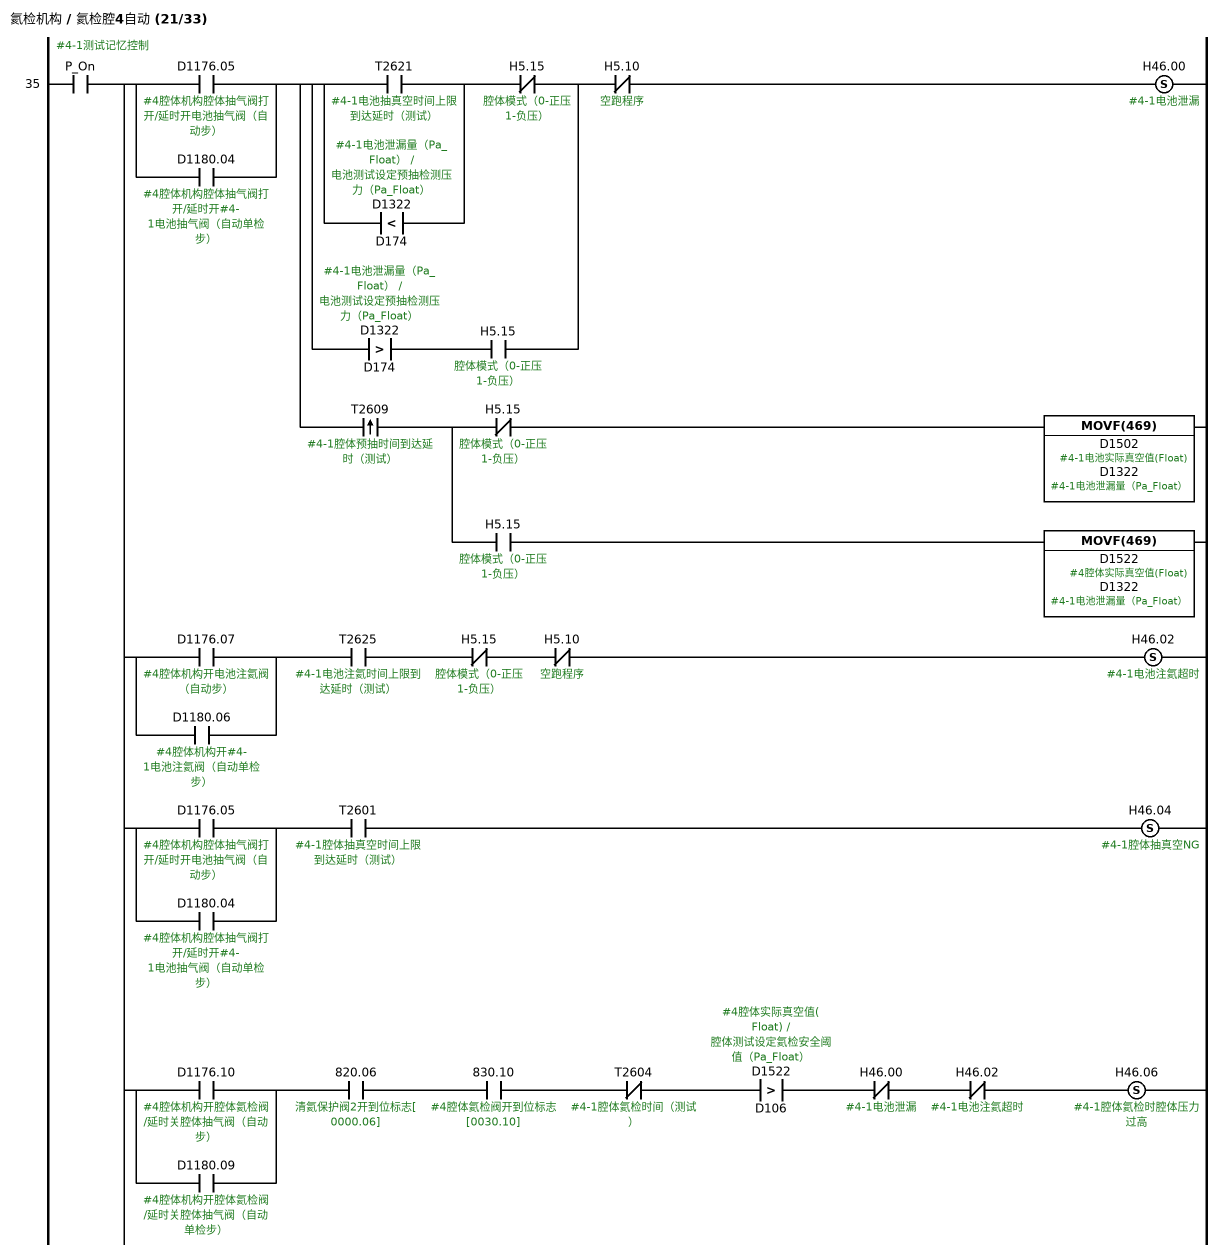
; [picture p360: 氦检机构 / 氦检腔4自动, rungs 35-35]

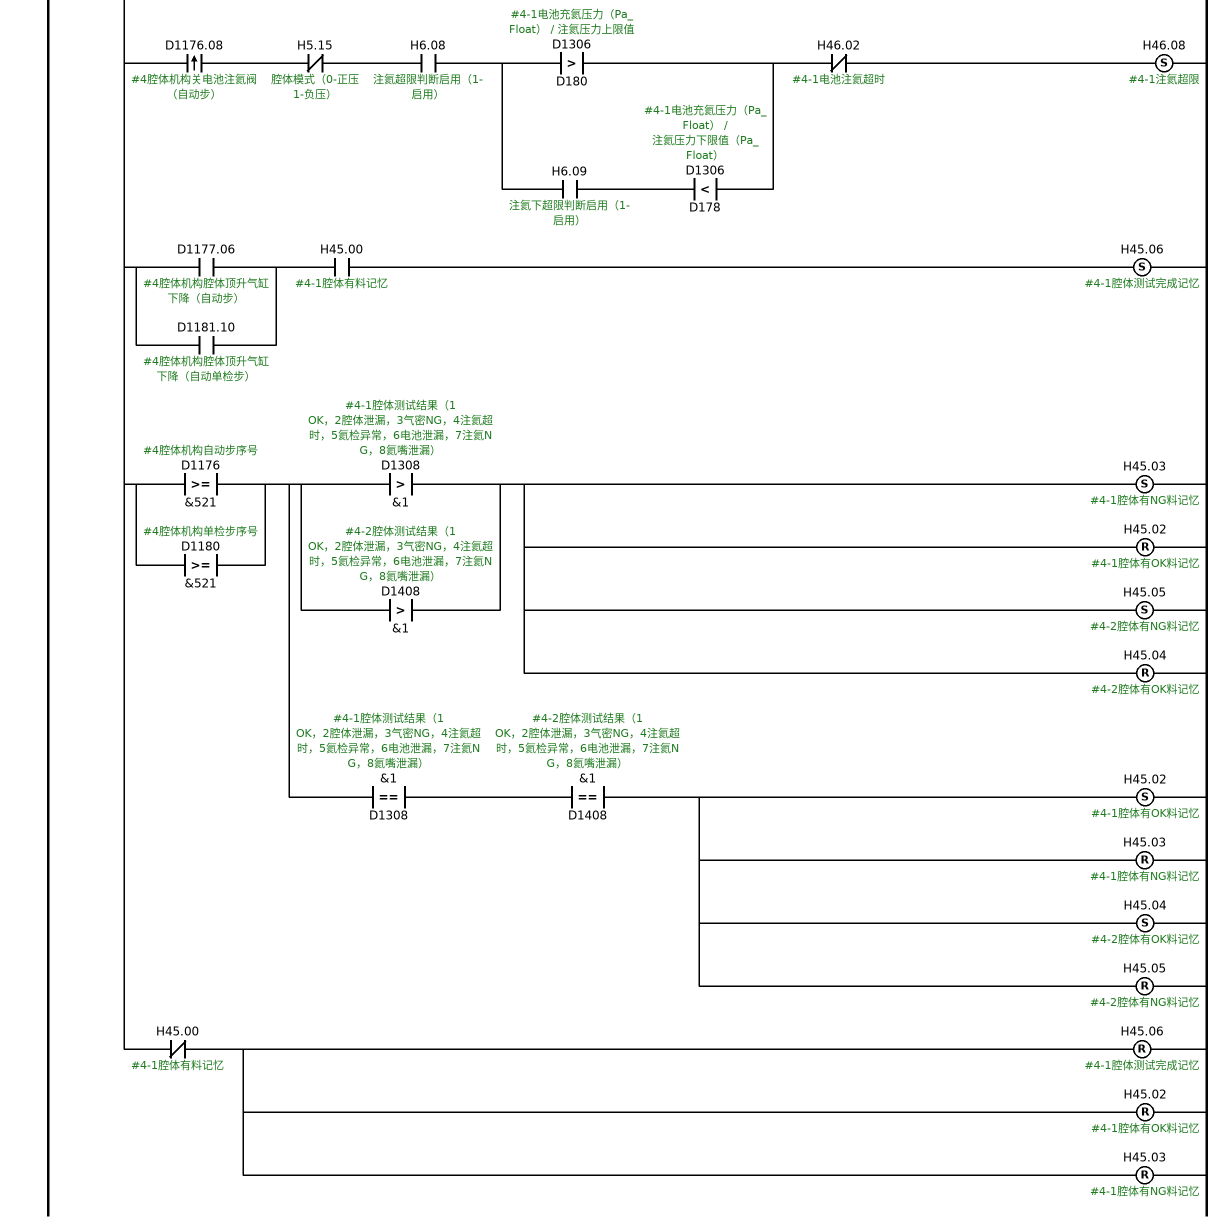
; rung 35: #4-1测试记忆控制
LD P_On
OUT TR0
LD D1176.05  ; #4腔体机构腔体抽气阀打开/延时开电池抽气阀（自动步）
OR D1180.04  ; #4腔体机构腔体抽气阀打开/延时开#4-1电池抽气阀（自动单检步）
ANDLD
OUT TR1
LD T2621  ; #4-1电池抽真空时间上限到达延时（测试）
OR<F(331) D1322 D174  ; #4-1电池泄漏量（Pa_Float）, 电池测试设定预抽检测压力（Pa_Float）
ANDNOT H5.15  ; 腔体模式（0-正压 1-负压）
LD>F(333) D1322 D174  ; #4-1电池泄漏量（Pa_Float）, 电池测试设定预抽检测压力（Pa_Float）
AND H5.15  ; 腔体模式（0-正压 1-负压）
ORLD
ANDLD
ANDNOT H5.10  ; 空跑程序
SET H46.00  ; #4-1电池泄漏
LD TR1
@AND T2609  ; #4-1腔体预抽时间到达延时（测试）
OUT TR1
ANDNOT H5.15  ; 腔体模式（0-正压 1-负压）
MOVF(469) D1502 D1322  ; #4-1电池实际真空值(Float), #4-1电池泄漏量（Pa_Float）
LD TR1
AND H5.15  ; 腔体模式（0-正压 1-负压）
MOVF(469) D1522 D1322  ; #4腔体实际真空值(Float), #4-1电池泄漏量（Pa_Float）
LD TR0
LD D1176.07  ; #4腔体机构开电池注氦阀（自动步）
OR D1180.06  ; #4腔体机构开#4-1电池注氦阀（自动单检步）
ANDLD
AND T2625  ; #4-1电池注氦时间上限到达延时（测试）
ANDNOT H5.15  ; 腔体模式（0-正压 1-负压）
ANDNOT H5.10  ; 空跑程序
SET H46.02  ; #4-1电池注氦超时
LD TR0
LD D1176.05  ; #4腔体机构腔体抽气阀打开/延时开电池抽气阀（自动步）
OR D1180.04  ; #4腔体机构腔体抽气阀打开/延时开#4-1电池抽气阀（自动单检步）
ANDLD
AND T2601  ; #4-1腔体抽真空时间上限到达延时（测试）
SET H46.04  ; #4-1腔体抽真空NG
LD TR0
LD D1176.10  ; #4腔体机构开腔体氦检阀/延时关腔体抽气阀（自动步）
OR D1180.09  ; #4腔体机构开腔体氦检阀/延时关腔体抽气阀（自动单检步）
ANDLD
AND 820.06  ; 清氦保护阀2开到位标志[0000.06]
AND 830.10  ; #4腔体氦检阀开到位标志[0030.10]
ANDNOT T2604  ; #4-1腔体氦检时间（测试）
AND>F(333) D1522 D106  ; #4腔体实际真空值(Float), 腔体测试设定氦检安全阈值（Pa_Float）
ANDNOT H46.00  ; #4-1电池泄漏
ANDNOT H46.02  ; #4-1电池注氦超时
SET H46.06  ; #4-1腔体氦检时腔体压力过高
LD TR0
@AND D1176.08  ; #4腔体机构关电池注氦阀（自动步）
ANDNOT H5.15  ; 腔体模式（0-正压 1-负压）
AND H6.08  ; 注氦超限判断启用（1-启用）
LD>F(333) D1306 D180  ; #4-1电池充氦压力（Pa_Float）, 注氦压力上限值
LD H6.09  ; 注氦下超限判断启用（1-启用）
AND<F(331) D1306 D178  ; #4-1电池充氦压力（Pa_Float）, 注氦压力下限值（Pa_Float）
ORLD
ANDLD
ANDNOT H46.02  ; #4-1电池注氦超时
SET H46.08  ; #4-1注氦超限
LD TR0
LD D1177.06  ; #4腔体机构腔体顶升气缸下降（自动步）
OR D1181.10  ; #4腔体机构腔体顶升气缸下降（自动单检步）
ANDLD
AND H45.00  ; #4-1腔体有料记忆
SET H45.06  ; #4-1腔体测试完成记忆
LD TR0
LD>=L(326) D1176 &521  ; #4腔体机构自动步序号
OR>=L(326) D1180 &521  ; #4腔体机构单检步序号
ANDLD
OUT TR1
LD>(320) D1308 &1  ; #4-1腔体测试结果（1 OK，2腔体泄漏，3气密NG，4注氦超时，5氦检异常，6电池泄漏，7注氦NG，8氦嘴泄漏）
OR>(320) D1408 &1  ; #4-2腔体测试结果（1 OK，2腔体泄漏，3气密NG，4注氦超时，5氦检异常，6电池泄漏，7注氦NG，8氦嘴泄漏）
ANDLD
SET H45.03  ; #4-1腔体有NG料记忆
RSET H45.02  ; #4-1腔体有OK料记忆
SET H45.05  ; #4-2腔体有NG料记忆
RSET H45.04  ; #4-2腔体有OK料记忆
LD TR1
AND=(300) &1 D1308  ; #4-1腔体测试结果（1 OK，2腔体泄漏，3气密NG，4注氦超时，5氦检异常，6电池泄漏，7注氦NG，8氦嘴泄漏）
AND=(300) &1 D1408  ; #4-2腔体测试结果（1 OK，2腔体泄漏，3气密NG，4注氦超时，5氦检异常，6电池泄漏，7注氦NG，8氦嘴泄漏）
SET H45.02  ; #4-1腔体有OK料记忆
RSET H45.03  ; #4-1腔体有NG料记忆
SET H45.04  ; #4-2腔体有OK料记忆
RSET H45.05  ; #4-2腔体有NG料记忆
LD TR0
ANDNOT H45.00  ; #4-1腔体有料记忆
RSET H45.06  ; #4-1腔体测试完成记忆
RSET H45.02  ; #4-1腔体有OK料记忆
RSET H45.03  ; #4-1腔体有NG料记忆

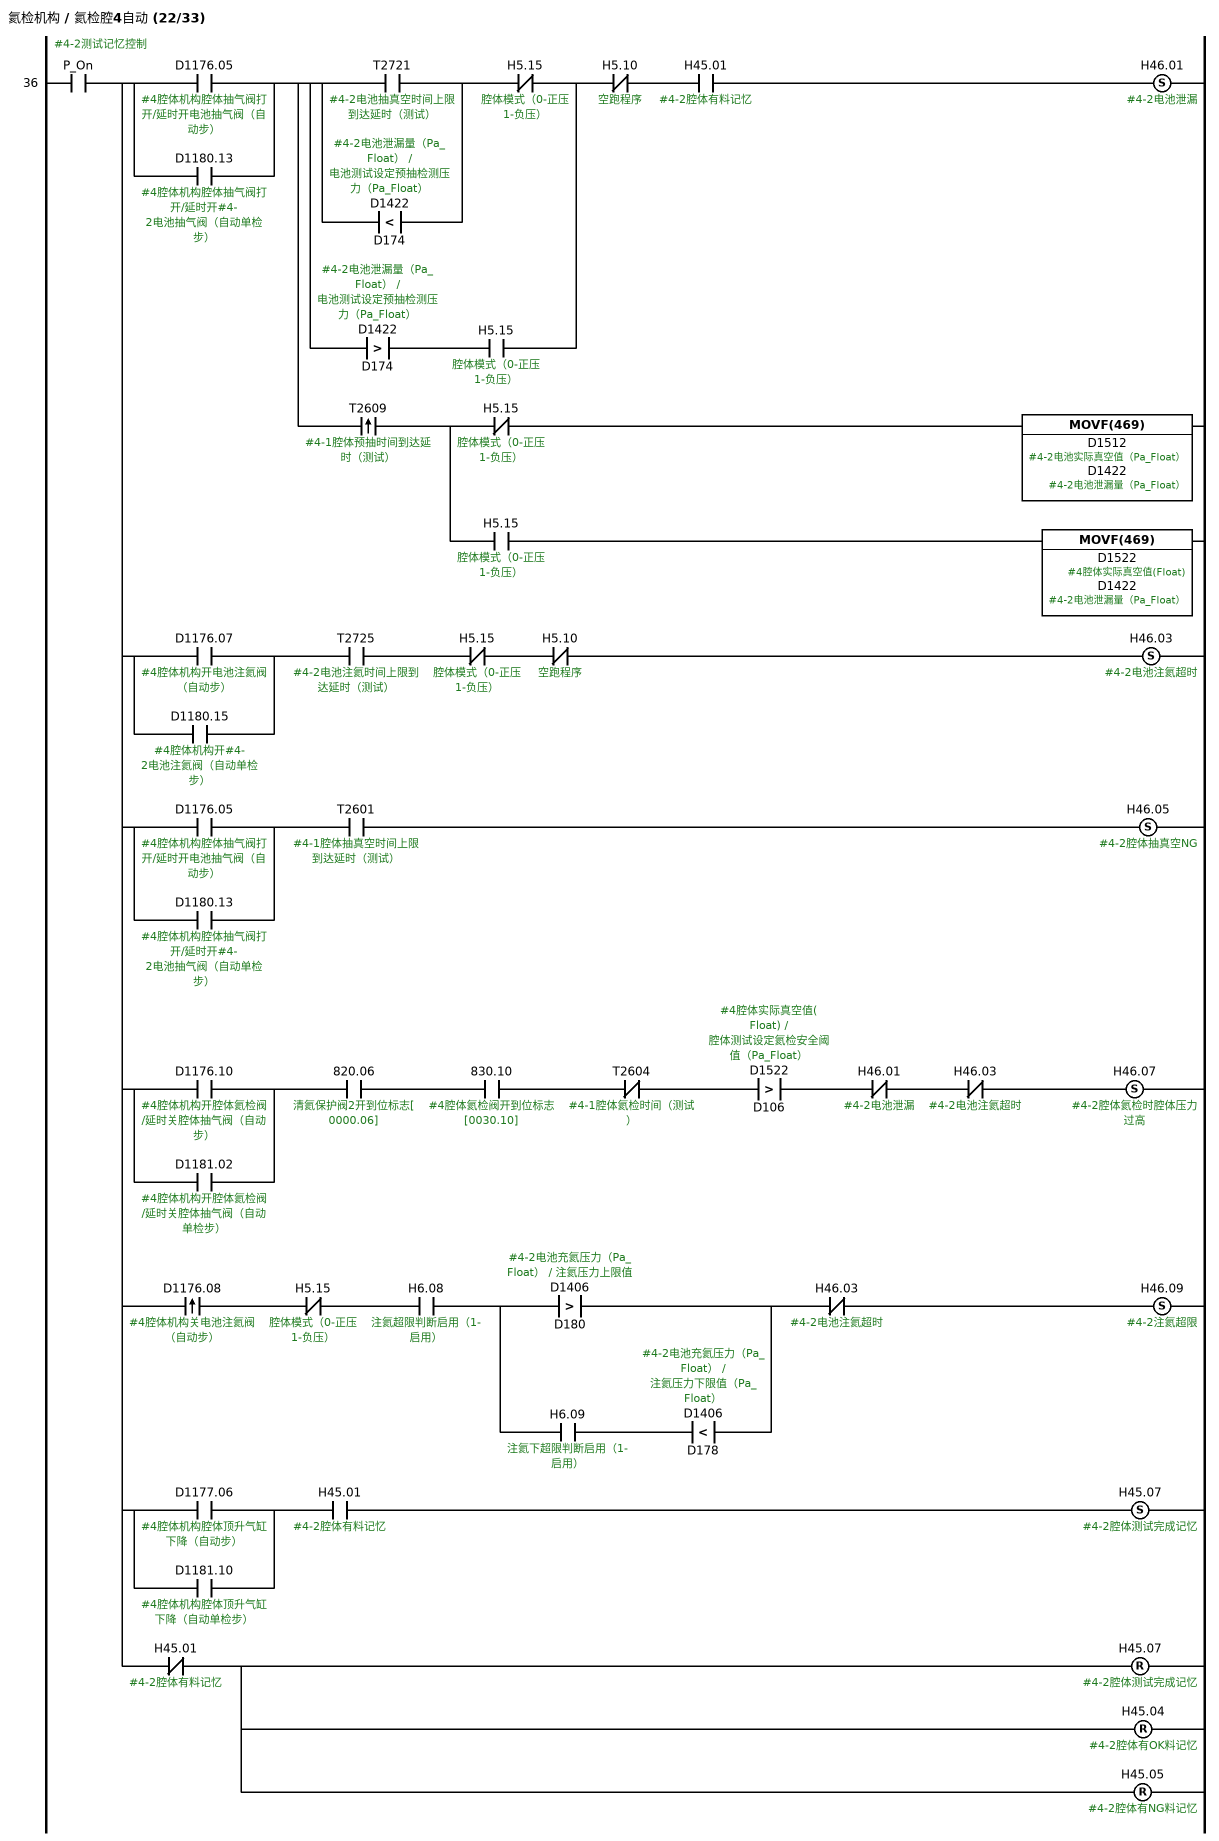
; rung 36: #4-2测试记忆控制
LD P_On
OUT TR0
LD D1176.05  ; #4腔体机构腔体抽气阀打开/延时开电池抽气阀（自动步）
OR D1180.13  ; #4腔体机构腔体抽气阀打开/延时开#4-2电池抽气阀（自动单检步）
ANDLD
OUT TR1
LD T2721  ; #4-2电池抽真空时间上限到达延时（测试）
OR<F(331) D1422 D174  ; #4-2电池泄漏量（Pa_Float）, 电池测试设定预抽检测压力（Pa_Float）
ANDNOT H5.15  ; 腔体模式（0-正压 1-负压）
LD>F(333) D1422 D174  ; #4-2电池泄漏量（Pa_Float）, 电池测试设定预抽检测压力（Pa_Float）
AND H5.15  ; 腔体模式（0-正压 1-负压）
ORLD
ANDLD
ANDNOT H5.10  ; 空跑程序
AND H45.01  ; #4-2腔体有料记忆
SET H46.01  ; #4-2电池泄漏
LD TR1
@AND T2609  ; #4-1腔体预抽时间到达延时（测试）
OUT TR1
ANDNOT H5.15  ; 腔体模式（0-正压 1-负压）
MOVF(469) D1512 D1422  ; #4-2电池实际真空值（Pa_Float）, #4-2电池泄漏量（Pa_Float）
LD TR1
AND H5.15  ; 腔体模式（0-正压 1-负压）
MOVF(469) D1522 D1422  ; #4腔体实际真空值(Float), #4-2电池泄漏量（Pa_Float）
LD TR0
LD D1176.07  ; #4腔体机构开电池注氦阀（自动步）
OR D1180.15  ; #4腔体机构开#4-2电池注氦阀（自动单检步）
ANDLD
AND T2725  ; #4-2电池注氦时间上限到达延时（测试）
ANDNOT H5.15  ; 腔体模式（0-正压 1-负压）
ANDNOT H5.10  ; 空跑程序
SET H46.03  ; #4-2电池注氦超时
LD TR0
LD D1176.05  ; #4腔体机构腔体抽气阀打开/延时开电池抽气阀（自动步）
OR D1180.13  ; #4腔体机构腔体抽气阀打开/延时开#4-2电池抽气阀（自动单检步）
ANDLD
AND T2601  ; #4-1腔体抽真空时间上限到达延时（测试）
SET H46.05  ; #4-2腔体抽真空NG
LD TR0
LD D1176.10  ; #4腔体机构开腔体氦检阀/延时关腔体抽气阀（自动步）
OR D1181.02  ; #4腔体机构开腔体氦检阀/延时关腔体抽气阀（自动单检步）
ANDLD
AND 820.06  ; 清氦保护阀2开到位标志[0000.06]
AND 830.10  ; #4腔体氦检阀开到位标志[0030.10]
ANDNOT T2604  ; #4-1腔体氦检时间（测试）
AND>F(333) D1522 D106  ; #4腔体实际真空值(Float), 腔体测试设定氦检安全阈值（Pa_Float）
ANDNOT H46.01  ; #4-2电池泄漏
ANDNOT H46.03  ; #4-2电池注氦超时
SET H46.07  ; #4-2腔体氦检时腔体压力过高
LD TR0
@AND D1176.08  ; #4腔体机构关电池注氦阀（自动步）
ANDNOT H5.15  ; 腔体模式（0-正压 1-负压）
AND H6.08  ; 注氦超限判断启用（1-启用）
LD>F(333) D1406 D180  ; #4-2电池充氦压力（Pa_Float）, 注氦压力上限值
LD H6.09  ; 注氦下超限判断启用（1-启用）
AND<F(331) D1406 D178  ; #4-2电池充氦压力（Pa_Float）, 注氦压力下限值（Pa_Float）
ORLD
ANDLD
ANDNOT H46.03  ; #4-2电池注氦超时
SET H46.09  ; #4-2注氦超限
LD TR0
LD D1177.06  ; #4腔体机构腔体顶升气缸下降（自动步）
OR D1181.10  ; #4腔体机构腔体顶升气缸下降（自动单检步）
ANDLD
AND H45.01  ; #4-2腔体有料记忆
SET H45.07  ; #4-2腔体测试完成记忆
LD TR0
ANDNOT H45.01  ; #4-2腔体有料记忆
RSET H45.07  ; #4-2腔体测试完成记忆
RSET H45.04  ; #4-2腔体有OK料记忆
RSET H45.05  ; #4-2腔体有NG料记忆

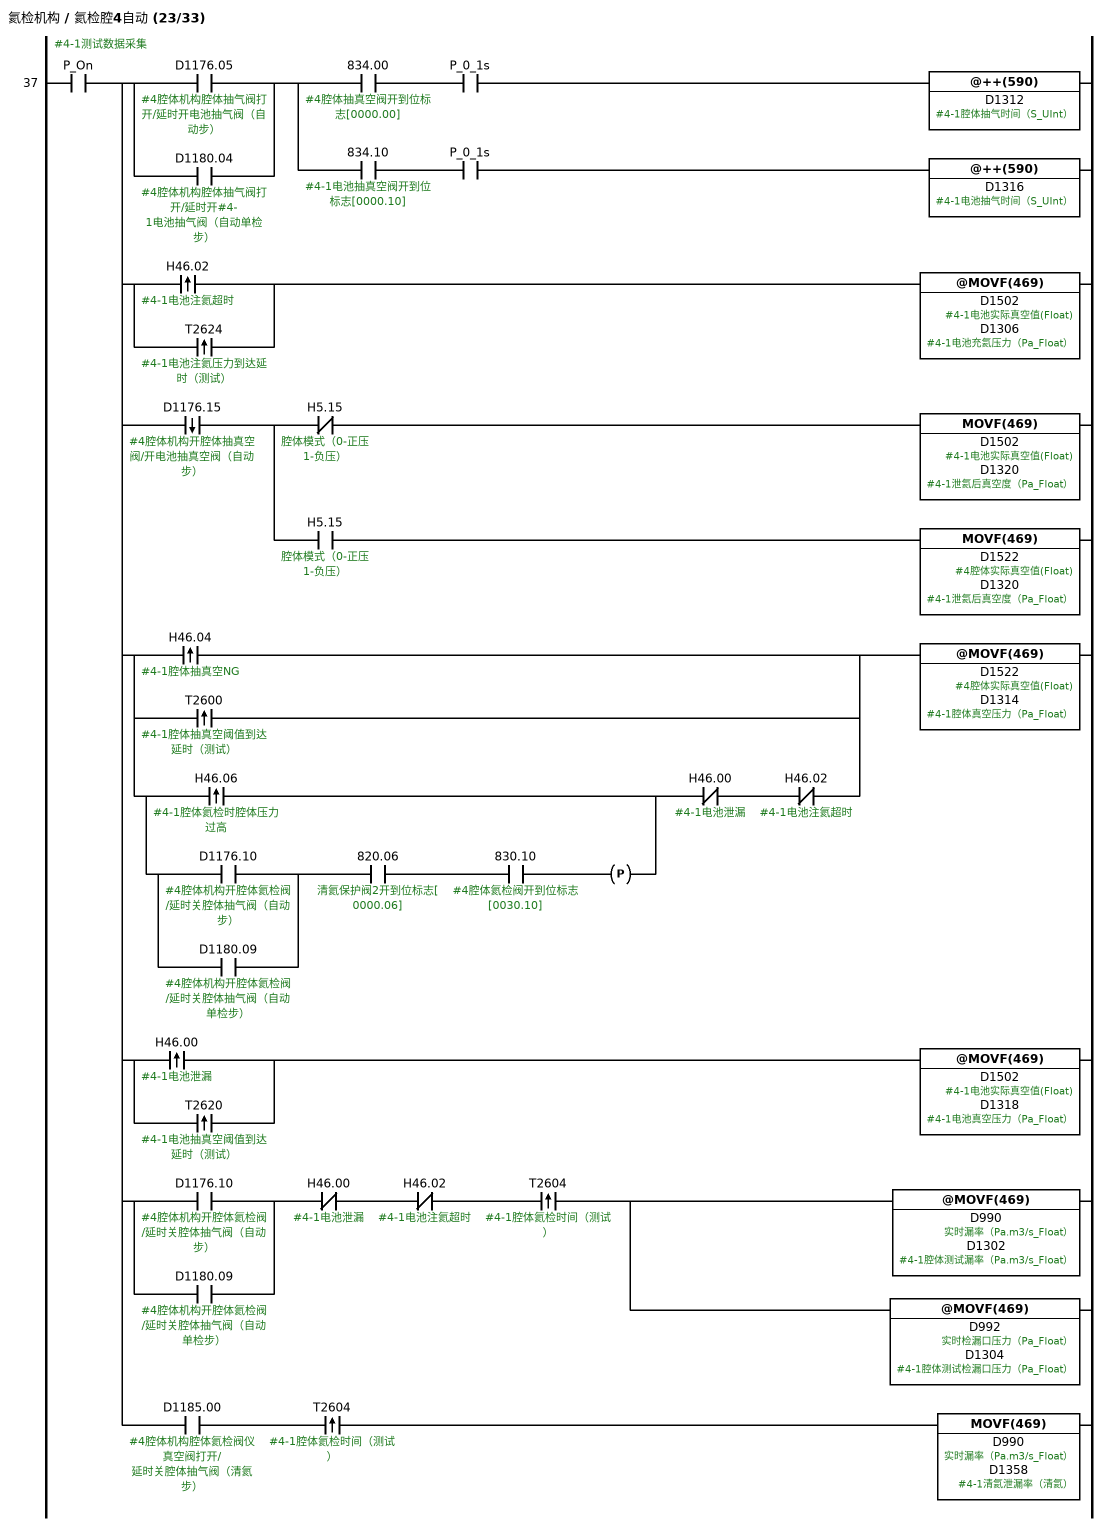
; rung 37: #4-1测试数据采集
LD P_On
OUT TR0
LD D1176.05  ; #4腔体机构腔体抽气阀打开/延时开电池抽气阀（自动步）
OR D1180.04  ; #4腔体机构腔体抽气阀打开/延时开#4-1电池抽气阀（自动单检步）
ANDLD
OUT TR1
AND 834.00  ; #4腔体抽真空阀开到位标志[0000.00]
AND P_0_1s
@++(590) D1312  ; #4-1腔体抽气时间（S_UInt）
LD TR1
AND 834.10  ; #4-1电池抽真空阀开到位标志[0000.10]
AND P_0_1s
@++(590) D1316  ; #4-1电池抽气时间（S_UInt）
LD TR0
@LD H46.02  ; #4-1电池注氦超时
@OR T2624  ; #4-1电池注氦压力到达延时（测试）
ANDLD
@MOVF(469) D1502 D1306  ; #4-1电池实际真空值(Float), #4-1电池充氦压力（Pa_Float）
LD TR0
%AND D1176.15  ; #4腔体机构开腔体抽真空阀/开电池抽真空阀（自动步）
OUT TR1
ANDNOT H5.15  ; 腔体模式（0-正压 1-负压）
MOVF(469) D1502 D1320  ; #4-1电池实际真空值(Float), #4-1泄氦后真空度（Pa_Float）
LD TR1
AND H5.15  ; 腔体模式（0-正压 1-负压）
MOVF(469) D1522 D1320  ; #4腔体实际真空值(Float), #4-1泄氦后真空度（Pa_Float）
LD TR0
@LD H46.04  ; #4-1腔体抽真空NG
@OR T2600  ; #4-1腔体抽真空阈值到达延时（测试）
@LD H46.06  ; #4-1腔体氦检时腔体压力过高
LD D1176.10  ; #4腔体机构开腔体氦检阀/延时关腔体抽气阀（自动步）
OR D1180.09  ; #4腔体机构开腔体氦检阀/延时关腔体抽气阀（自动单检步）
AND 820.06  ; 清氦保护阀2开到位标志[0000.06]
AND 830.10  ; #4腔体氦检阀开到位标志[0030.10]
UP(521)
ORLD
ANDNOT H46.00  ; #4-1电池泄漏
ANDNOT H46.02  ; #4-1电池注氦超时
ORLD
ANDLD
@MOVF(469) D1522 D1314  ; #4腔体实际真空值(Float), #4-1腔体真空压力（Pa_Float）
LD TR0
@LD H46.00  ; #4-1电池泄漏
@OR T2620  ; #4-1电池抽真空阈值到达延时（测试）
ANDLD
@MOVF(469) D1502 D1318  ; #4-1电池实际真空值(Float), #4-1电池真空压力（Pa_Float）
LD TR0
LD D1176.10  ; #4腔体机构开腔体氦检阀/延时关腔体抽气阀（自动步）
OR D1180.09  ; #4腔体机构开腔体氦检阀/延时关腔体抽气阀（自动单检步）
ANDLD
ANDNOT H46.00  ; #4-1电池泄漏
ANDNOT H46.02  ; #4-1电池注氦超时
@AND T2604  ; #4-1腔体氦检时间（测试）
@MOVF(469) D990 D1302  ; 实时漏率（Pa.m3/s_Float）, #4-1腔体测试漏率（Pa.m3/s_Float）
@MOVF(469) D992 D1304  ; 实时检漏口压力（Pa_Float）, #4-1腔体测试检漏口压力（Pa_Float）
LD TR0
AND D1185.00  ; #4腔体机构腔体氦检阀仪真空阀打开/延时关腔体抽气阀（清氦步）
@AND T2604  ; #4-1腔体氦检时间（测试）
MOVF(469) D990 D1358  ; 实时漏率（Pa.m3/s_Float）, #4-1清氦泄漏率（清氦）

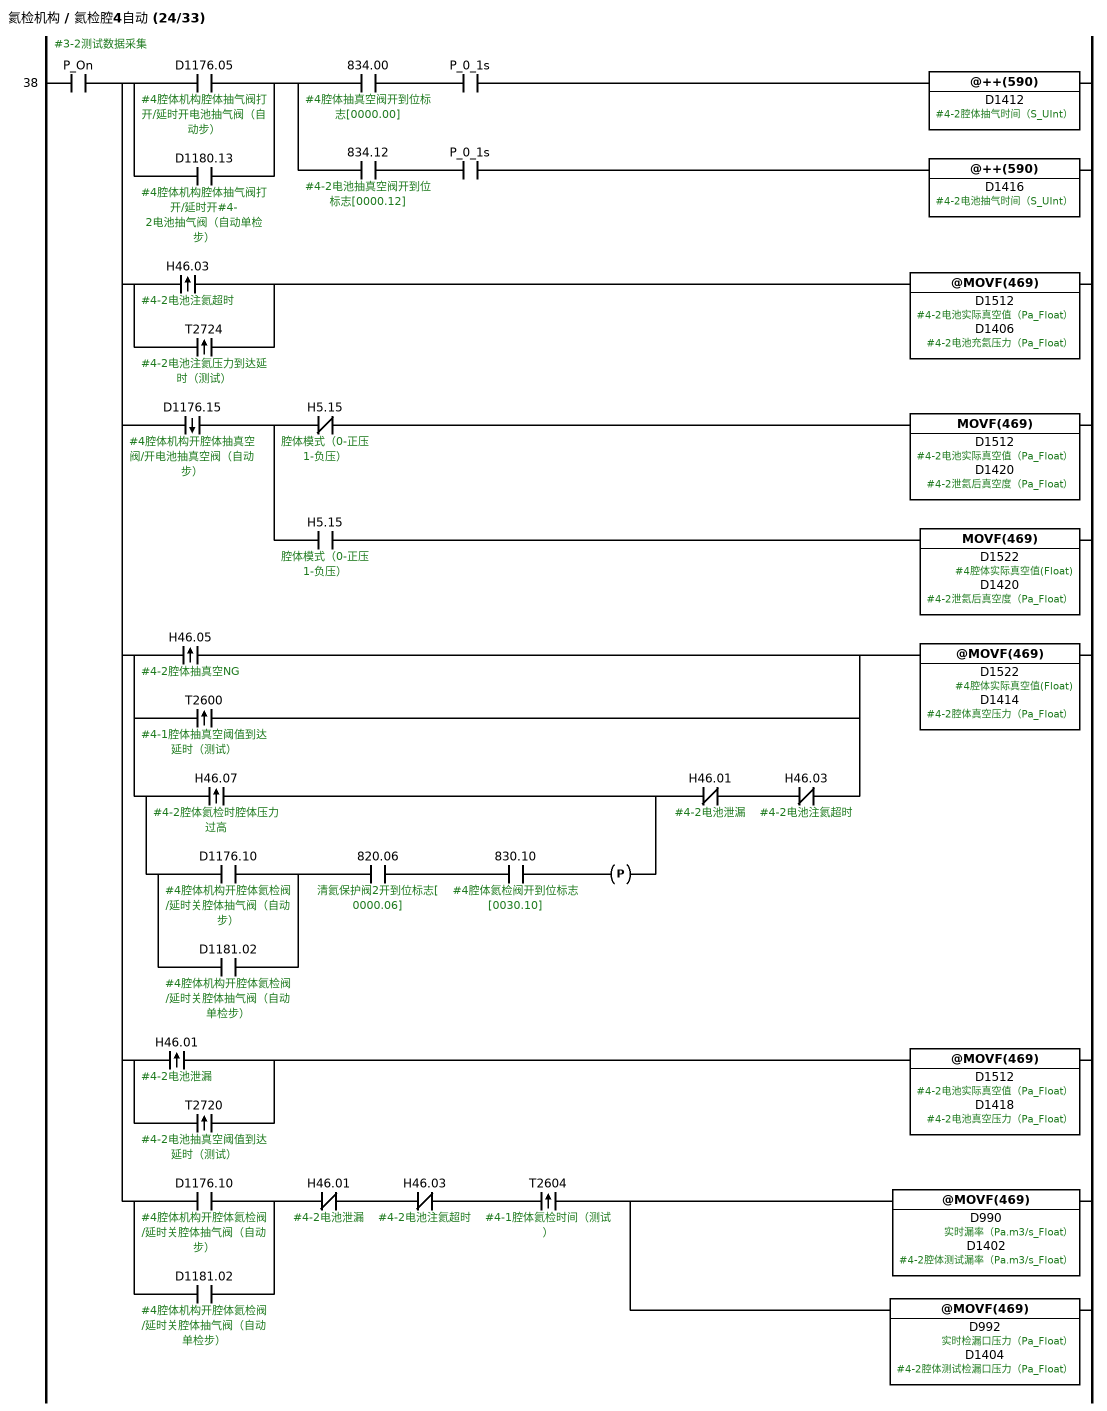
; rung 38: #3-2测试数据采集
LD P_On
OUT TR0
LD D1176.05  ; #4腔体机构腔体抽气阀打开/延时开电池抽气阀（自动步）
OR D1180.13  ; #4腔体机构腔体抽气阀打开/延时开#4-2电池抽气阀（自动单检步）
ANDLD
OUT TR1
AND 834.00  ; #4腔体抽真空阀开到位标志[0000.00]
AND P_0_1s
@++(590) D1412  ; #4-2腔体抽气时间（S_UInt）
LD TR1
AND 834.12  ; #4-2电池抽真空阀开到位标志[0000.12]
AND P_0_1s
@++(590) D1416  ; #4-2电池抽气时间（S_UInt）
LD TR0
@LD H46.03  ; #4-2电池注氦超时
@OR T2724  ; #4-2电池注氦压力到达延时（测试）
ANDLD
@MOVF(469) D1512 D1406  ; #4-2电池实际真空值（Pa_Float）, #4-2电池充氦压力（Pa_Float）
LD TR0
%AND D1176.15  ; #4腔体机构开腔体抽真空阀/开电池抽真空阀（自动步）
OUT TR1
ANDNOT H5.15  ; 腔体模式（0-正压 1-负压）
MOVF(469) D1512 D1420  ; #4-2电池实际真空值（Pa_Float）, #4-2泄氦后真空度（Pa_Float）
LD TR1
AND H5.15  ; 腔体模式（0-正压 1-负压）
MOVF(469) D1522 D1420  ; #4腔体实际真空值(Float), #4-2泄氦后真空度（Pa_Float）
LD TR0
@LD H46.05  ; #4-2腔体抽真空NG
@OR T2600  ; #4-1腔体抽真空阈值到达延时（测试）
@LD H46.07  ; #4-2腔体氦检时腔体压力过高
LD D1176.10  ; #4腔体机构开腔体氦检阀/延时关腔体抽气阀（自动步）
OR D1181.02  ; #4腔体机构开腔体氦检阀/延时关腔体抽气阀（自动单检步）
AND 820.06  ; 清氦保护阀2开到位标志[0000.06]
AND 830.10  ; #4腔体氦检阀开到位标志[0030.10]
UP(521)
ORLD
ANDNOT H46.01  ; #4-2电池泄漏
ANDNOT H46.03  ; #4-2电池注氦超时
ORLD
ANDLD
@MOVF(469) D1522 D1414  ; #4腔体实际真空值(Float), #4-2腔体真空压力（Pa_Float）
LD TR0
@LD H46.01  ; #4-2电池泄漏
@OR T2720  ; #4-2电池抽真空阈值到达延时（测试）
ANDLD
@MOVF(469) D1512 D1418  ; #4-2电池实际真空值（Pa_Float）, #4-2电池真空压力（Pa_Float）
LD TR0
LD D1176.10  ; #4腔体机构开腔体氦检阀/延时关腔体抽气阀（自动步）
OR D1181.02  ; #4腔体机构开腔体氦检阀/延时关腔体抽气阀（自动单检步）
ANDLD
ANDNOT H46.01  ; #4-2电池泄漏
ANDNOT H46.03  ; #4-2电池注氦超时
@AND T2604  ; #4-1腔体氦检时间（测试）
@MOVF(469) D990 D1402  ; 实时漏率（Pa.m3/s_Float）, #4-2腔体测试漏率（Pa.m3/s_Float）
@MOVF(469) D992 D1404  ; 实时检漏口压力（Pa_Float）, #4-2腔体测试检漏口压力（Pa_Float）

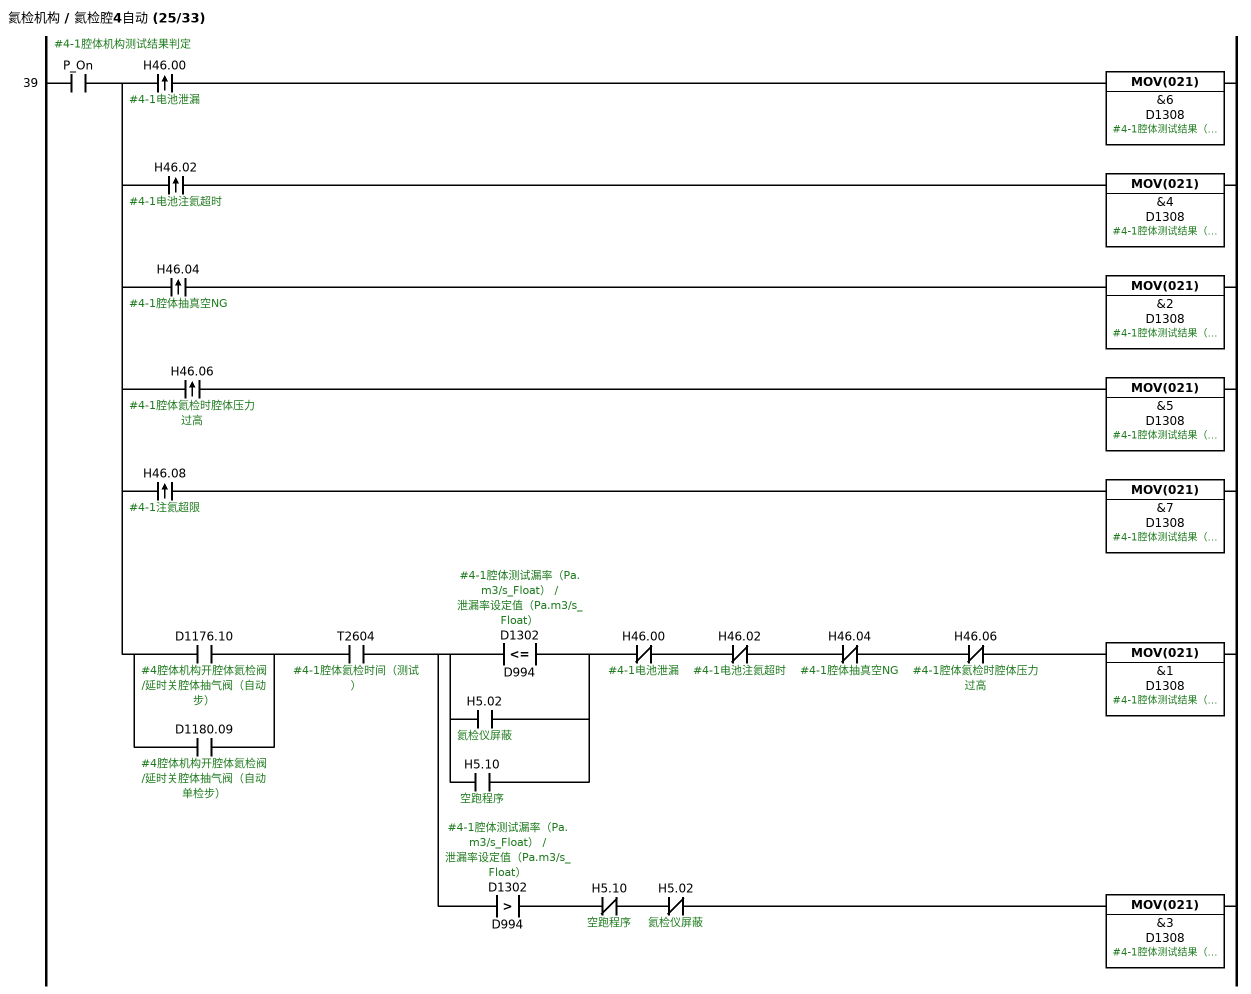
; rung 39: #4-1腔体机构测试结果判定
LD P_On
OUT TR0
@AND H46.00  ; #4-1电池泄漏
MOV(021) &6 D1308  ; #4-1腔体测试结果（1 OK，2腔体泄漏，3气密NG，4注氦超时，5氦检异常，6电池泄漏，7注氦NG，8氦嘴泄漏）
LD TR0
@AND H46.02  ; #4-1电池注氦超时
MOV(021) &4 D1308  ; #4-1腔体测试结果（1 OK，2腔体泄漏，3气密NG，4注氦超时，5氦检异常，6电池泄漏，7注氦NG，8氦嘴泄漏）
LD TR0
@AND H46.04  ; #4-1腔体抽真空NG
MOV(021) &2 D1308  ; #4-1腔体测试结果（1 OK，2腔体泄漏，3气密NG，4注氦超时，5氦检异常，6电池泄漏，7注氦NG，8氦嘴泄漏）
LD TR0
@AND H46.06  ; #4-1腔体氦检时腔体压力过高
MOV(021) &5 D1308  ; #4-1腔体测试结果（1 OK，2腔体泄漏，3气密NG，4注氦超时，5氦检异常，6电池泄漏，7注氦NG，8氦嘴泄漏）
LD TR0
@AND H46.08  ; #4-1注氦超限
MOV(021) &7 D1308  ; #4-1腔体测试结果（1 OK，2腔体泄漏，3气密NG，4注氦超时，5氦检异常，6电池泄漏，7注氦NG，8氦嘴泄漏）
LD TR0
LD D1176.10  ; #4腔体机构开腔体氦检阀/延时关腔体抽气阀（自动步）
OR D1180.09  ; #4腔体机构开腔体氦检阀/延时关腔体抽气阀（自动单检步）
ANDLD
AND T2604  ; #4-1腔体氦检时间（测试）
OUT TR0
LD<=F(332) D1302 D994  ; #4-1腔体测试漏率（Pa.m3/s_Float）, 泄漏率设定值（Pa.m3/s_Float）
OR H5.02  ; 氦检仪屏蔽
OR H5.10  ; 空跑程序
ANDLD
ANDNOT H46.00  ; #4-1电池泄漏
ANDNOT H46.02  ; #4-1电池注氦超时
ANDNOT H46.04  ; #4-1腔体抽真空NG
ANDNOT H46.06  ; #4-1腔体氦检时腔体压力过高
MOV(021) &1 D1308  ; #4-1腔体测试结果（1 OK，2腔体泄漏，3气密NG，4注氦超时，5氦检异常，6电池泄漏，7注氦NG，8氦嘴泄漏）
LD TR0
AND>F(333) D1302 D994  ; #4-1腔体测试漏率（Pa.m3/s_Float）, 泄漏率设定值（Pa.m3/s_Float）
ANDNOT H5.10  ; 空跑程序
ANDNOT H5.02  ; 氦检仪屏蔽
MOV(021) &3 D1308  ; #4-1腔体测试结果（1 OK，2腔体泄漏，3气密NG，4注氦超时，5氦检异常，6电池泄漏，7注氦NG，8氦嘴泄漏）

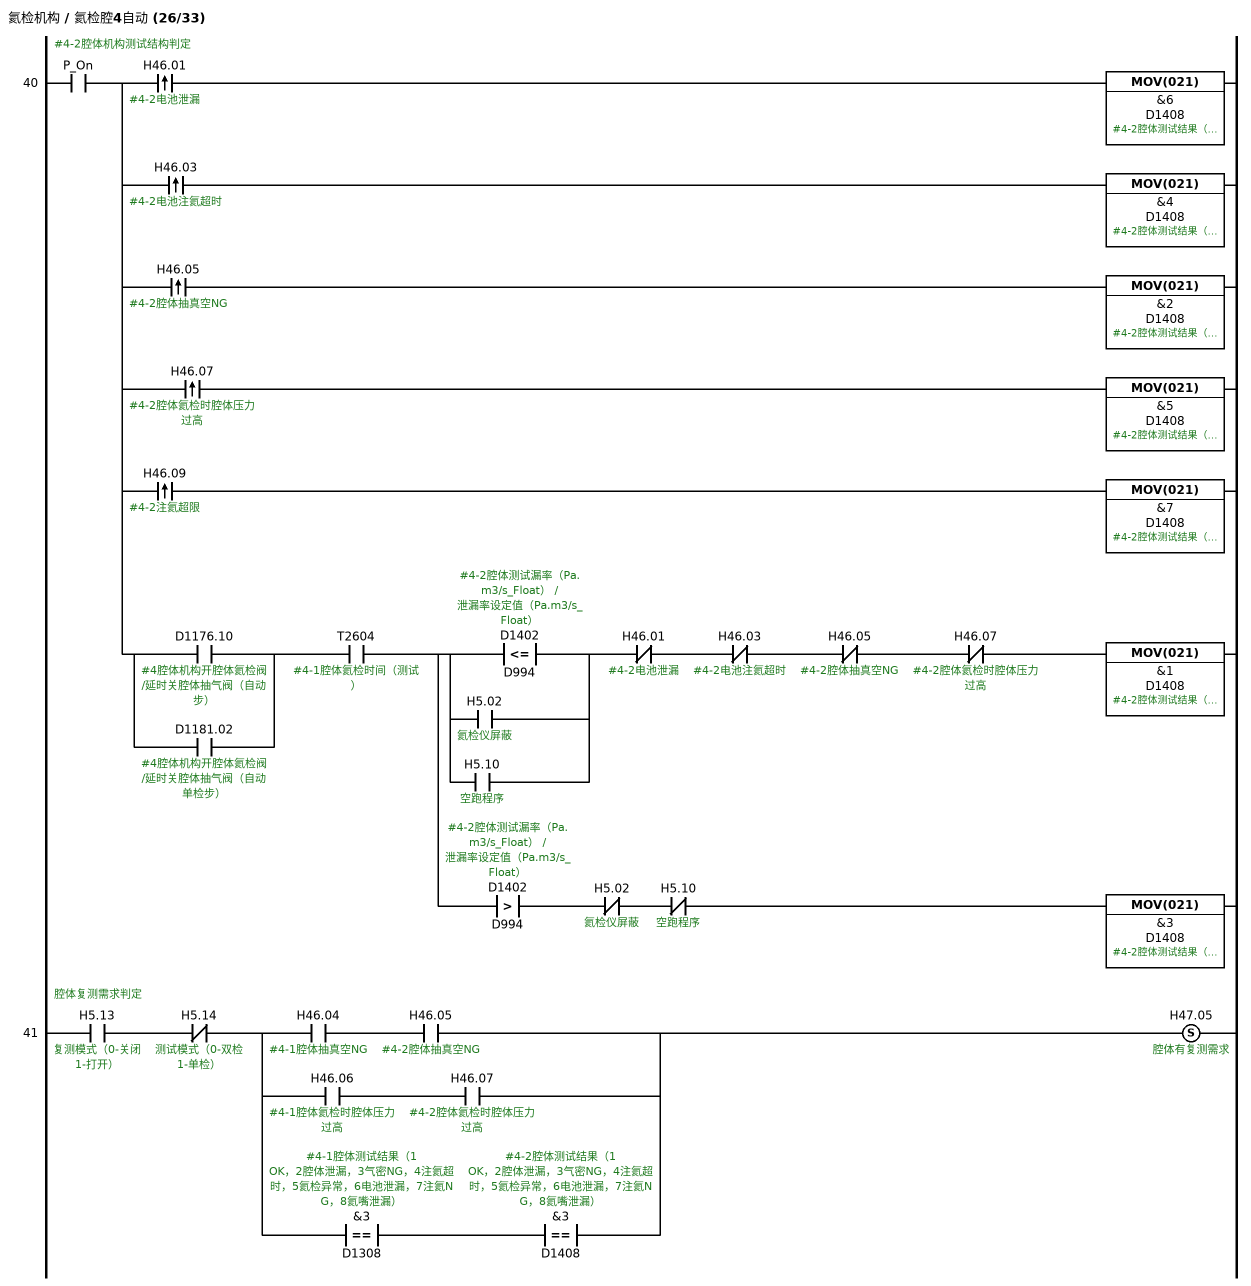
; rung 40: #4-2腔体机构测试结构判定
LD P_On
OUT TR0
@AND H46.01  ; #4-2电池泄漏
MOV(021) &6 D1408  ; #4-2腔体测试结果（1 OK，2腔体泄漏，3气密NG，4注氦超时，5氦检异常，6电池泄漏，7注氦NG，8氦嘴泄漏）
LD TR0
@AND H46.03  ; #4-2电池注氦超时
MOV(021) &4 D1408  ; #4-2腔体测试结果（1 OK，2腔体泄漏，3气密NG，4注氦超时，5氦检异常，6电池泄漏，7注氦NG，8氦嘴泄漏）
LD TR0
@AND H46.05  ; #4-2腔体抽真空NG
MOV(021) &2 D1408  ; #4-2腔体测试结果（1 OK，2腔体泄漏，3气密NG，4注氦超时，5氦检异常，6电池泄漏，7注氦NG，8氦嘴泄漏）
LD TR0
@AND H46.07  ; #4-2腔体氦检时腔体压力过高
MOV(021) &5 D1408  ; #4-2腔体测试结果（1 OK，2腔体泄漏，3气密NG，4注氦超时，5氦检异常，6电池泄漏，7注氦NG，8氦嘴泄漏）
LD TR0
@AND H46.09  ; #4-2注氦超限
MOV(021) &7 D1408  ; #4-2腔体测试结果（1 OK，2腔体泄漏，3气密NG，4注氦超时，5氦检异常，6电池泄漏，7注氦NG，8氦嘴泄漏）
LD TR0
LD D1176.10  ; #4腔体机构开腔体氦检阀/延时关腔体抽气阀（自动步）
OR D1181.02  ; #4腔体机构开腔体氦检阀/延时关腔体抽气阀（自动单检步）
ANDLD
AND T2604  ; #4-1腔体氦检时间（测试）
OUT TR0
LD<=F(332) D1402 D994  ; #4-2腔体测试漏率（Pa.m3/s_Float）, 泄漏率设定值（Pa.m3/s_Float）
OR H5.02  ; 氦检仪屏蔽
OR H5.10  ; 空跑程序
ANDLD
ANDNOT H46.01  ; #4-2电池泄漏
ANDNOT H46.03  ; #4-2电池注氦超时
ANDNOT H46.05  ; #4-2腔体抽真空NG
ANDNOT H46.07  ; #4-2腔体氦检时腔体压力过高
MOV(021) &1 D1408  ; #4-2腔体测试结果（1 OK，2腔体泄漏，3气密NG，4注氦超时，5氦检异常，6电池泄漏，7注氦NG，8氦嘴泄漏）
LD TR0
AND>F(333) D1402 D994  ; #4-2腔体测试漏率（Pa.m3/s_Float）, 泄漏率设定值（Pa.m3/s_Float）
ANDNOT H5.02  ; 氦检仪屏蔽
ANDNOT H5.10  ; 空跑程序
MOV(021) &3 D1408  ; #4-2腔体测试结果（1 OK，2腔体泄漏，3气密NG，4注氦超时，5氦检异常，6电池泄漏，7注氦NG，8氦嘴泄漏）
; rung 41: 腔体复测需求判定
LD H5.13  ; 复测模式（0-关闭 1-打开）
ANDNOT H5.14  ; 测试模式（0-双检 1-单检）
LD H46.04  ; #4-1腔体抽真空NG
AND H46.05  ; #4-2腔体抽真空NG
LD H46.06  ; #4-1腔体氦检时腔体压力过高
AND H46.07  ; #4-2腔体氦检时腔体压力过高
ORLD
LD=(300) &3 D1308  ; #4-1腔体测试结果（1 OK，2腔体泄漏，3气密NG，4注氦超时，5氦检异常，6电池泄漏，7注氦NG，8氦嘴泄漏）
AND=(300) &3 D1408  ; #4-2腔体测试结果（1 OK，2腔体泄漏，3气密NG，4注氦超时，5氦检异常，6电池泄漏，7注氦NG，8氦嘴泄漏）
ORLD
ANDLD
SET H47.05  ; 腔体有复测需求

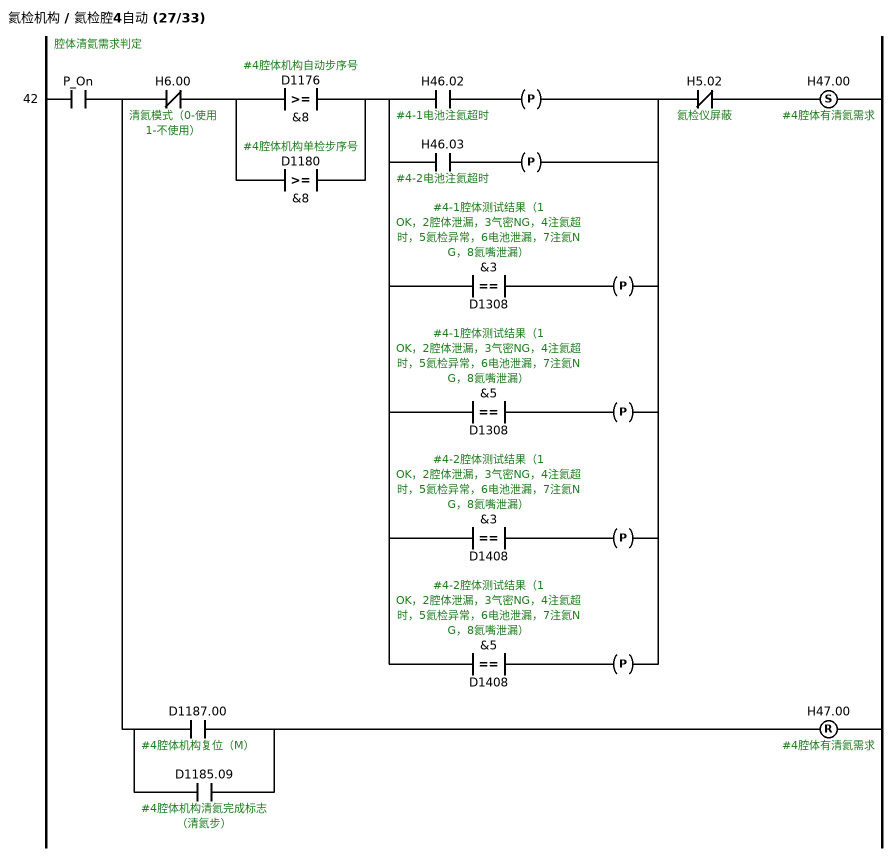
; rung 42: 腔体清氦需求判定
LD P_On
OUT TR0
ANDNOT H6.00  ; 清氦模式（0-使用 1-不使用）
LD>=L(326) D1176 &8  ; #4腔体机构自动步序号
OR>=L(326) D1180 &8  ; #4腔体机构单检步序号
ANDLD
LD H46.02  ; #4-1电池注氦超时
UP(521)
LD H46.03  ; #4-2电池注氦超时
UP(521)
ORLD
LD=(300) &3 D1308  ; #4-1腔体测试结果（1 OK，2腔体泄漏，3气密NG，4注氦超时，5氦检异常，6电池泄漏，7注氦NG，8氦嘴泄漏）
UP(521)
ORLD
LD=(300) &5 D1308  ; #4-1腔体测试结果（1 OK，2腔体泄漏，3气密NG，4注氦超时，5氦检异常，6电池泄漏，7注氦NG，8氦嘴泄漏）
UP(521)
ORLD
LD=(300) &3 D1408  ; #4-2腔体测试结果（1 OK，2腔体泄漏，3气密NG，4注氦超时，5氦检异常，6电池泄漏，7注氦NG，8氦嘴泄漏）
UP(521)
ORLD
LD=(300) &5 D1408  ; #4-2腔体测试结果（1 OK，2腔体泄漏，3气密NG，4注氦超时，5氦检异常，6电池泄漏，7注氦NG，8氦嘴泄漏）
UP(521)
ORLD
ANDLD
ANDNOT H5.02  ; 氦检仪屏蔽
SET H47.00  ; #4腔体有清氦需求
LD TR0
LD D1187.00  ; #4腔体机构复位（M）
OR D1185.09  ; #4腔体机构清氦完成标志（清氦步）
ANDLD
RSET H47.00  ; #4腔体有清氦需求

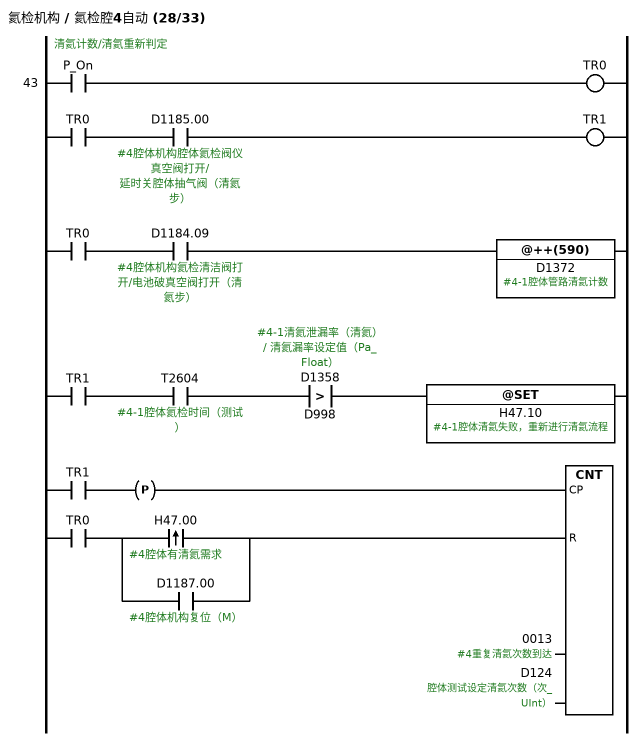
; rung 43: 清氦计数/清氦重新判定
LD P_On
OUT TR0
AND D1184.09  ; #4腔体机构氦检清洁阀打开/电池破真空阀打开（清氦步）
@++(590) D1372  ; #4-1腔体管路清氦计数
LD TR0
AND D1185.00  ; #4腔体机构腔体氦检阀仪真空阀打开/延时关腔体抽气阀（清氦步）
OUT TR1
AND T2604  ; #4-1腔体氦检时间（测试）
AND>F(333) D1358 D998  ; #4-1清氦泄漏率（清氦）, 清氦漏率设定值（Pa_Float）
@SET H47.10  ; #4-1腔体清氦失败，重新进行清氦流程
LD TR1
UP(521)
LD TR0
@LD H47.00  ; #4腔体有清氦需求
OR D1187.00  ; #4腔体机构复位（M）
ANDLD
CNT 0013 D124  ; 腔体测试设定清氦次数（次_UInt）, #4重复清氦次数到达

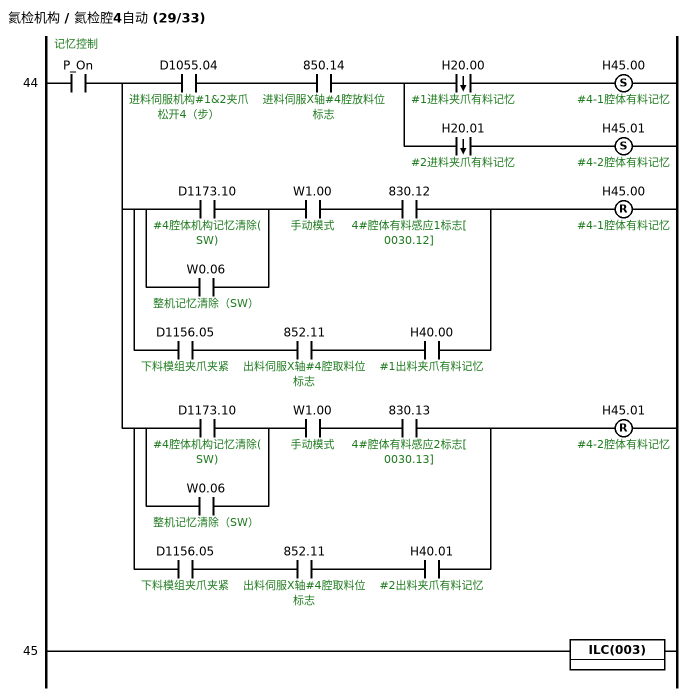
; rung 44: 记忆控制
LD P_On
OUT TR0
AND D1055.04  ; 进料伺服机构#1&2夹爪松开4（步）
AND 850.14  ; 进料伺服X轴#4腔放料位标志
OUT TR1
%AND H20.00  ; #1进料夹爪有料记忆
SET H45.00  ; #4-1腔体有料记忆
LD TR1
%AND H20.01  ; #2进料夹爪有料记忆
SET H45.01  ; #4-2腔体有料记忆
LD TR0
LD D1173.10  ; #4腔体机构记忆清除(SW)
OR W0.06  ; 整机记忆清除（SW）
AND W1.00  ; 手动模式
AND 830.12  ; 4#腔体有料感应1标志[0030.12]
LD D1156.05  ; 下料模组夹爪夹紧
AND 852.11  ; 出料伺服X轴#4腔取料位标志
AND H40.00  ; #1出料夹爪有料记忆
ORLD
ANDLD
RSET H45.00  ; #4-1腔体有料记忆
LD TR0
LD D1173.10  ; #4腔体机构记忆清除(SW)
OR W0.06  ; 整机记忆清除（SW）
AND W1.00  ; 手动模式
AND 830.13  ; 4#腔体有料感应2标志[0030.13]
LD D1156.05  ; 下料模组夹爪夹紧
AND 852.11  ; 出料伺服X轴#4腔取料位标志
AND H40.01  ; #2出料夹爪有料记忆
ORLD
ANDLD
RSET H45.01  ; #4-2腔体有料记忆
; rung 45
ILC(003)

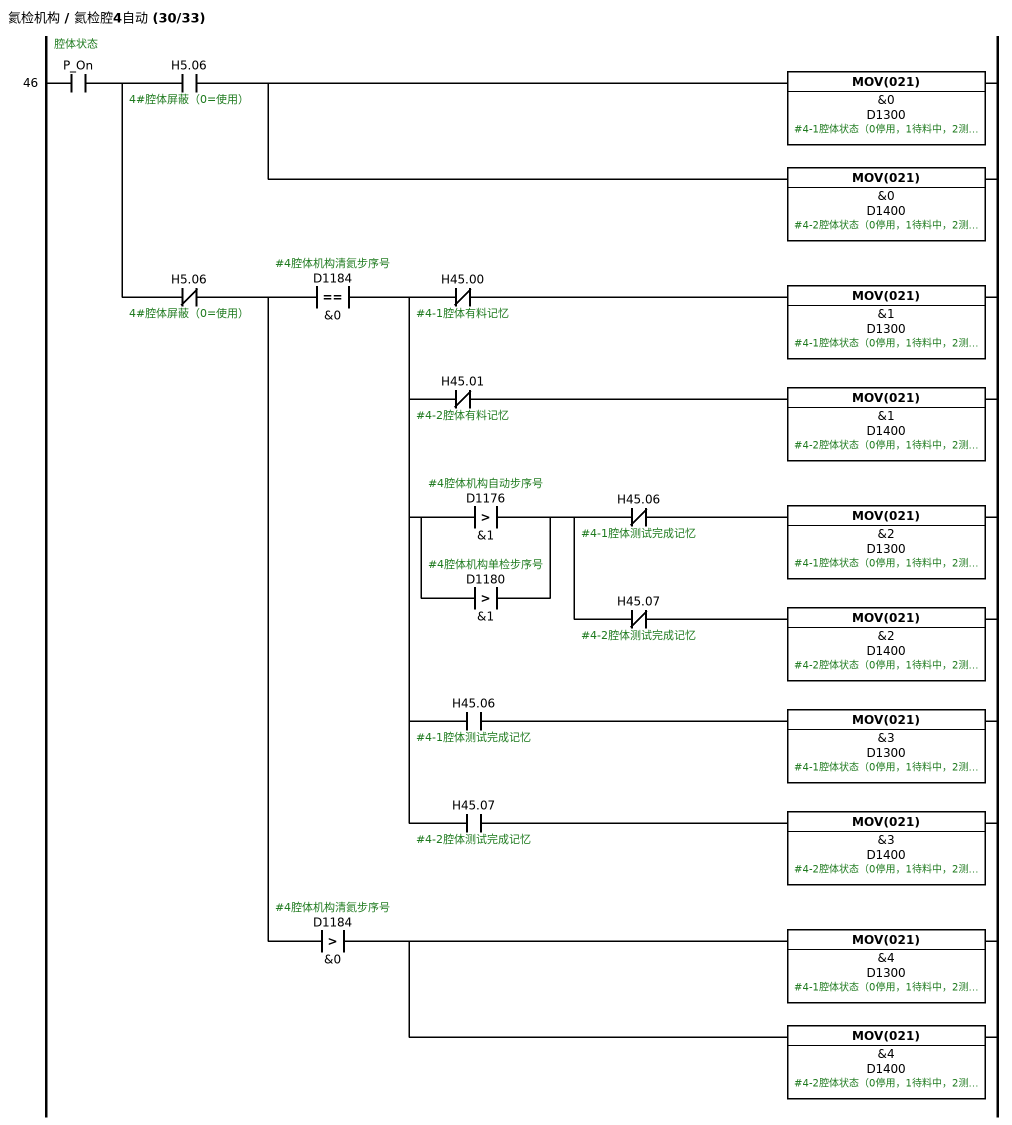
; rung 46: 腔体状态
LD P_On
OUT TR0
AND H5.06  ; 4#腔体屏蔽（0=使用）
MOV(021) &0 D1300  ; #4-1腔体状态（0停用，1待料中，2测试中，3测试完成）
MOV(021) &0 D1400  ; #4-2腔体状态（0停用，1待料中，2测试中，3测试完成）
LD TR0
ANDNOT H5.06  ; 4#腔体屏蔽（0=使用）
OUT TR0
AND=L(301) D1184 &0  ; #4腔体机构清氦步序号
OUT TR1
ANDNOT H45.00  ; #4-1腔体有料记忆
MOV(021) &1 D1300  ; #4-1腔体状态（0停用，1待料中，2测试中，3测试完成）
LD TR1
ANDNOT H45.01  ; #4-2腔体有料记忆
MOV(021) &1 D1400  ; #4-2腔体状态（0停用，1待料中，2测试中，3测试完成）
LD TR1
LD>L(321) D1176 &1  ; #4腔体机构自动步序号
OR>L(321) D1180 &1  ; #4腔体机构单检步序号
ANDLD
OUT TR2
ANDNOT H45.06  ; #4-1腔体测试完成记忆
MOV(021) &2 D1300  ; #4-1腔体状态（0停用，1待料中，2测试中，3测试完成）
LD TR2
ANDNOT H45.07  ; #4-2腔体测试完成记忆
MOV(021) &2 D1400  ; #4-2腔体状态（0停用，1待料中，2测试中，3测试完成）
LD TR1
AND H45.06  ; #4-1腔体测试完成记忆
MOV(021) &3 D1300  ; #4-1腔体状态（0停用，1待料中，2测试中，3测试完成）
LD TR1
AND H45.07  ; #4-2腔体测试完成记忆
MOV(021) &3 D1400  ; #4-2腔体状态（0停用，1待料中，2测试中，3测试完成）
LD TR0
AND>L(321) D1184 &0  ; #4腔体机构清氦步序号
MOV(021) &4 D1300  ; #4-1腔体状态（0停用，1待料中，2测试中，3测试完成）
MOV(021) &4 D1400  ; #4-2腔体状态（0停用，1待料中，2测试中，3测试完成）

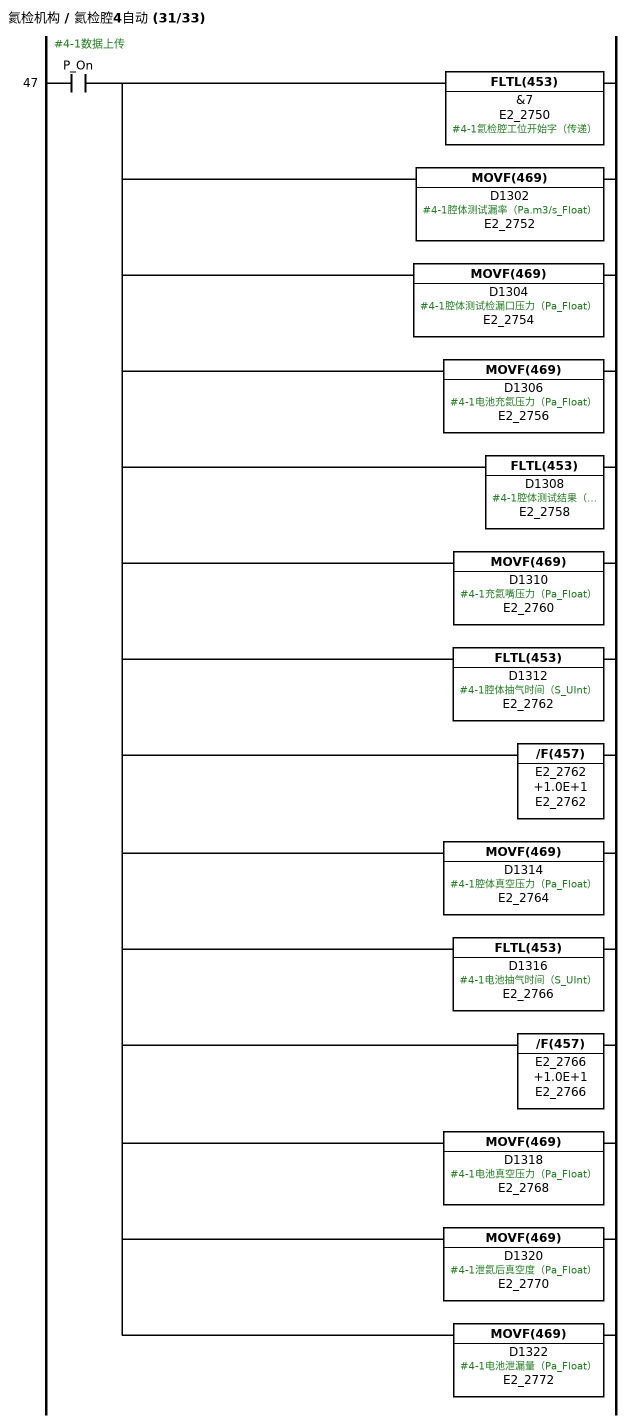
; rung 47: #4-1数据上传
LD P_On
FLTL(453) &7 E2_2750  ; #4-1氦检腔工位开始字（传递）
MOVF(469) D1302 E2_2752  ; #4-1腔体测试漏率（Pa.m3/s_Float）
MOVF(469) D1304 E2_2754  ; #4-1腔体测试检漏口压力（Pa_Float）
MOVF(469) D1306 E2_2756  ; #4-1电池充氦压力（Pa_Float）
FLTL(453) D1308 E2_2758  ; #4-1腔体测试结果（1 OK，2腔体泄漏，3气密NG，4注氦超时，5氦检异常，6电池泄漏，7注氦NG，8氦嘴泄漏）
MOVF(469) D1310 E2_2760  ; #4-1充氦嘴压力（Pa_Float）
FLTL(453) D1312 E2_2762  ; #4-1腔体抽气时间（S_UInt）
/F(457) E2_2762 +1.0E+1 E2_2762
MOVF(469) D1314 E2_2764  ; #4-1腔体真空压力（Pa_Float）
FLTL(453) D1316 E2_2766  ; #4-1电池抽气时间（S_UInt）
/F(457) E2_2766 +1.0E+1 E2_2766
MOVF(469) D1318 E2_2768  ; #4-1电池真空压力（Pa_Float）
MOVF(469) D1320 E2_2770  ; #4-1泄氦后真空度（Pa_Float）
MOVF(469) D1322 E2_2772  ; #4-1电池泄漏量（Pa_Float）

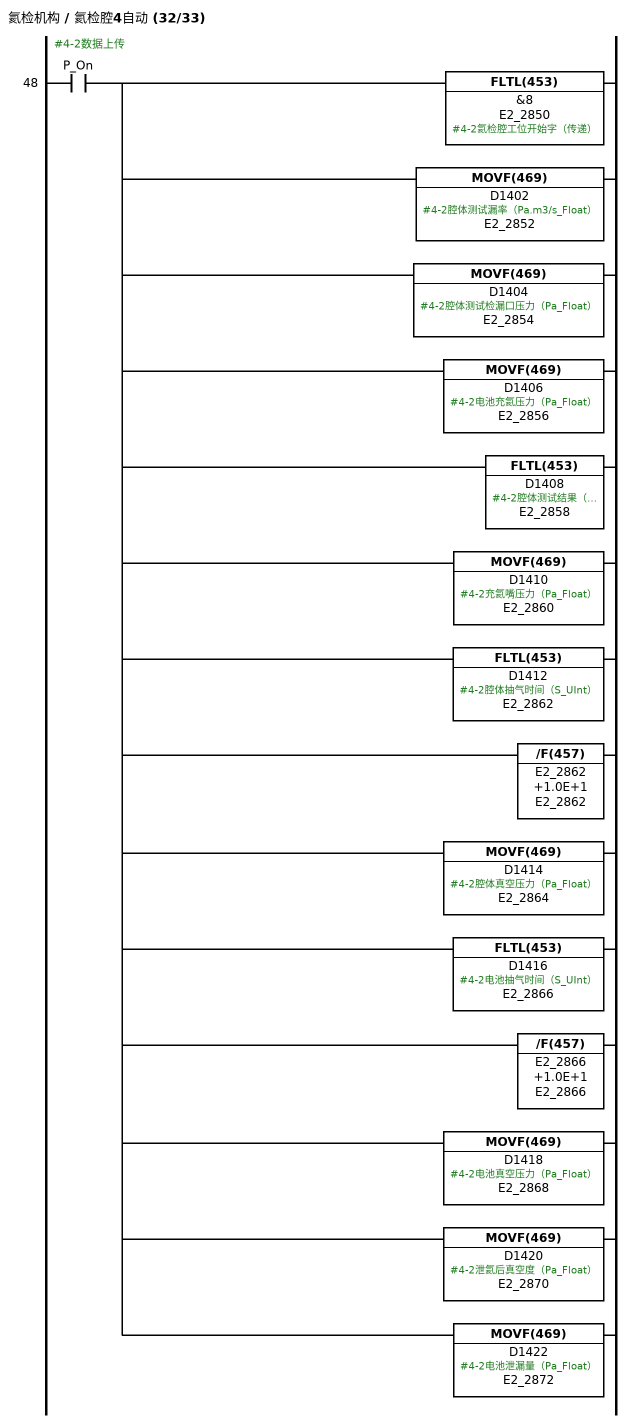
; rung 48: #4-2数据上传
LD P_On
FLTL(453) &8 E2_2850  ; #4-2氦检腔工位开始字（传递）
MOVF(469) D1402 E2_2852  ; #4-2腔体测试漏率（Pa.m3/s_Float）
MOVF(469) D1404 E2_2854  ; #4-2腔体测试检漏口压力（Pa_Float）
MOVF(469) D1406 E2_2856  ; #4-2电池充氦压力（Pa_Float）
FLTL(453) D1408 E2_2858  ; #4-2腔体测试结果（1 OK，2腔体泄漏，3气密NG，4注氦超时，5氦检异常，6电池泄漏，7注氦NG，8氦嘴泄漏）
MOVF(469) D1410 E2_2860  ; #4-2充氦嘴压力（Pa_Float）
FLTL(453) D1412 E2_2862  ; #4-2腔体抽气时间（S_UInt）
/F(457) E2_2862 +1.0E+1 E2_2862
MOVF(469) D1414 E2_2864  ; #4-2腔体真空压力（Pa_Float）
FLTL(453) D1416 E2_2866  ; #4-2电池抽气时间（S_UInt）
/F(457) E2_2866 +1.0E+1 E2_2866
MOVF(469) D1418 E2_2868  ; #4-2电池真空压力（Pa_Float）
MOVF(469) D1420 E2_2870  ; #4-2泄氦后真空度（Pa_Float）
MOVF(469) D1422 E2_2872  ; #4-2电池泄漏量（Pa_Float）

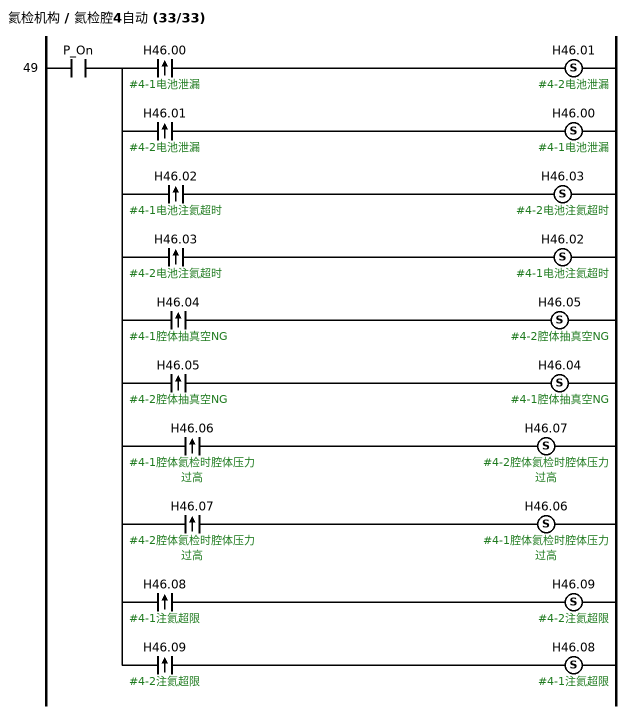
; rung 49
LD P_On
OUT TR0
@AND H46.00  ; #4-1电池泄漏
SET H46.01  ; #4-2电池泄漏
LD TR0
@AND H46.01  ; #4-2电池泄漏
SET H46.00  ; #4-1电池泄漏
LD TR0
@AND H46.02  ; #4-1电池注氦超时
SET H46.03  ; #4-2电池注氦超时
LD TR0
@AND H46.03  ; #4-2电池注氦超时
SET H46.02  ; #4-1电池注氦超时
LD TR0
@AND H46.04  ; #4-1腔体抽真空NG
SET H46.05  ; #4-2腔体抽真空NG
LD TR0
@AND H46.05  ; #4-2腔体抽真空NG
SET H46.04  ; #4-1腔体抽真空NG
LD TR0
@AND H46.06  ; #4-1腔体氦检时腔体压力过高
SET H46.07  ; #4-2腔体氦检时腔体压力过高
LD TR0
@AND H46.07  ; #4-2腔体氦检时腔体压力过高
SET H46.06  ; #4-1腔体氦检时腔体压力过高
LD TR0
@AND H46.08  ; #4-1注氦超限
SET H46.09  ; #4-2注氦超限
LD TR0
@AND H46.09  ; #4-2注氦超限
SET H46.08  ; #4-1注氦超限

### Section 工站复位

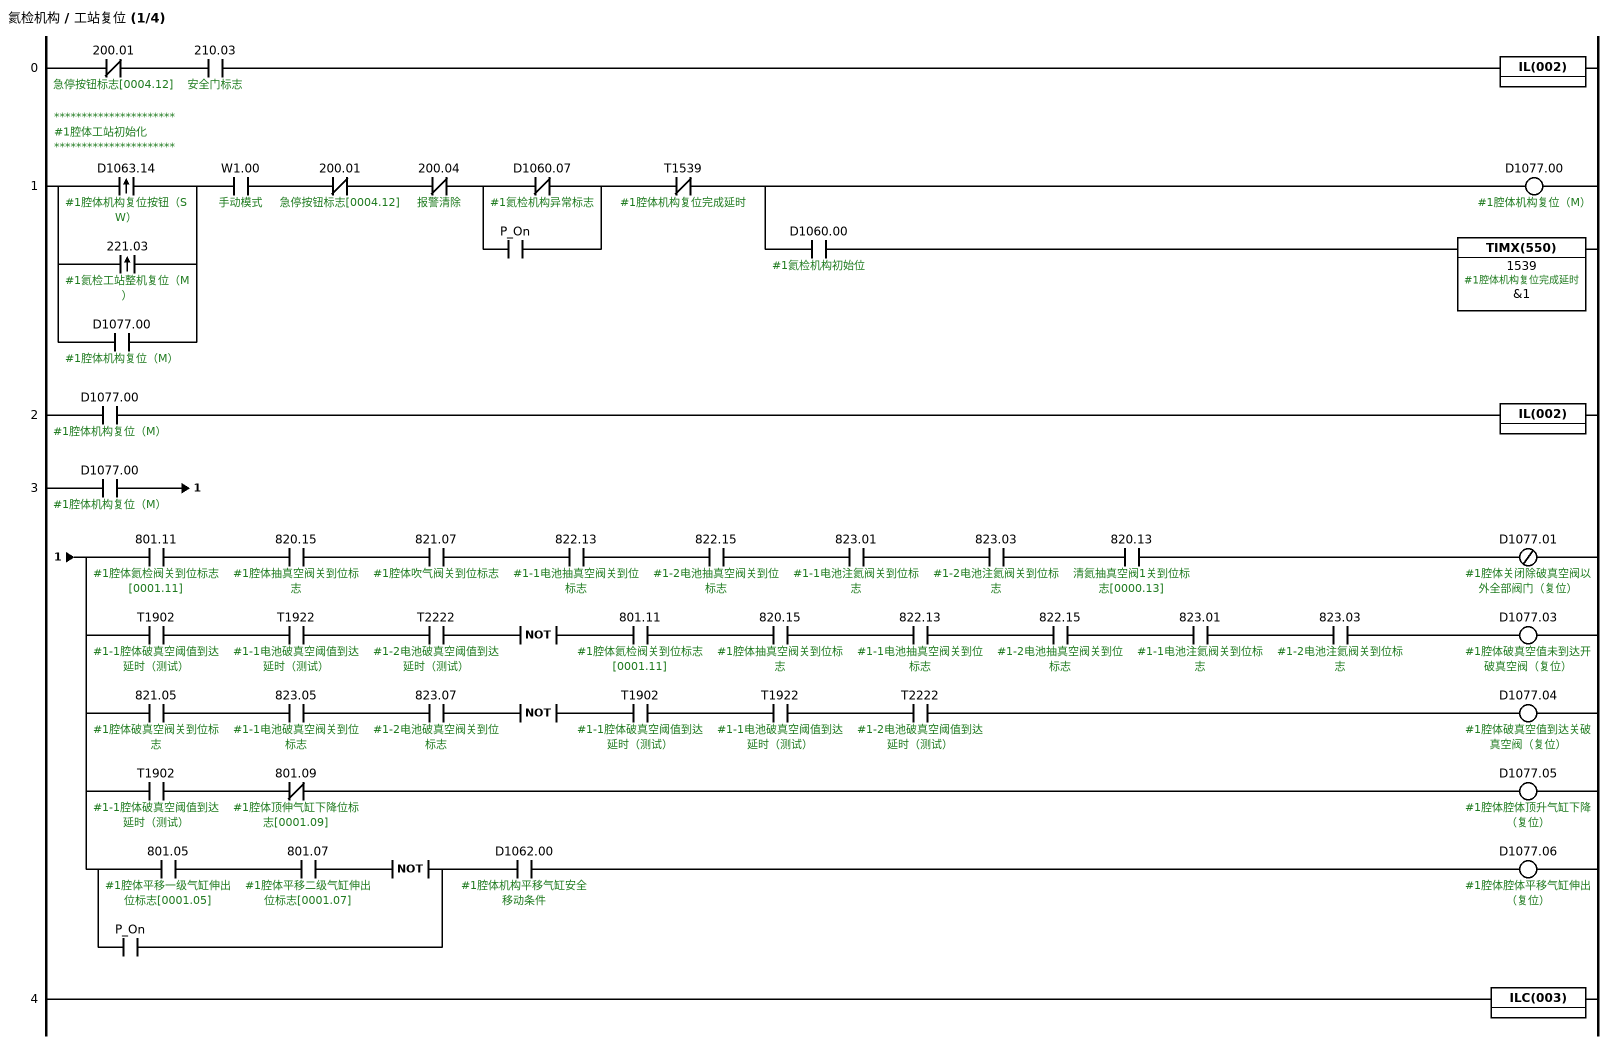
; rung 0
LDNOT 200.01  ; 急停按钮标志[0004.12]
AND 210.03  ; 安全门标志
IL(002)
; rung 1: ********************** / #1腔体工站初始化 / **********************
@LD D1063.14  ; #1腔体机构复位按钮（SW）
@OR 221.03  ; #1氦检工站整机复位（M）
OR D1077.00  ; #1腔体机构复位（M）
AND W1.00  ; 手动模式
ANDNOT 200.01  ; 急停按钮标志[0004.12]
ANDNOT 200.04  ; 报警清除
LDNOT D1060.07  ; #1氦检机构异常标志
OR P_On
ANDLD
ANDNOT T1539  ; #1腔体机构复位完成延时
OUT D1077.00  ; #1腔体机构复位（M）
AND D1060.00  ; #1氦检机构初始位
TIMX(550) 1539 &1  ; #1腔体机构复位完成延时
; rung 2
LD D1077.00  ; #1腔体机构复位（M）
IL(002)
; rung 3
LD D1077.00  ; #1腔体机构复位（M）
OUT TR0
AND 801.11  ; #1腔体氦检阀关到位标志[0001.11]
AND 820.15  ; #1腔体抽真空阀关到位标志
AND 821.07  ; #1腔体吹气阀关到位标志
AND 822.13  ; #1-1电池抽真空阀关到位标志
AND 822.15  ; #1-2电池抽真空阀关到位标志
AND 823.01  ; #1-1电池注氦阀关到位标志
AND 823.03  ; #1-2电池注氦阀关到位标志
AND 820.13  ; 清氦抽真空阀1关到位标志[0000.13]
OUTNOT D1077.01  ; #1腔体关闭除破真空阀以外全部阀门（复位）
LD TR0
AND T1902  ; #1-1腔体破真空阈值到达延时（测试）
AND T1922  ; #1-1电池破真空阈值到达延时（测试）
AND T2222  ; #1-2电池破真空阈值到达延时（测试）
NOT(520)
AND 801.11  ; #1腔体氦检阀关到位标志[0001.11]
AND 820.15  ; #1腔体抽真空阀关到位标志
AND 822.13  ; #1-1电池抽真空阀关到位标志
AND 822.15  ; #1-2电池抽真空阀关到位标志
AND 823.01  ; #1-1电池注氦阀关到位标志
AND 823.03  ; #1-2电池注氦阀关到位标志
OUT D1077.03  ; #1腔体破真空值未到达开破真空阀（复位）
LD TR0
AND 821.05  ; #1腔体破真空阀关到位标志
AND 823.05  ; #1-1电池破真空阀关到位标志
AND 823.07  ; #1-2电池破真空阀关到位标志
NOT(520)
AND T1902  ; #1-1腔体破真空阈值到达延时（测试）
AND T1922  ; #1-1电池破真空阈值到达延时（测试）
AND T2222  ; #1-2电池破真空阈值到达延时（测试）
OUT D1077.04  ; #1腔体破真空值到达关破真空阀（复位）
LD TR0
AND T1902  ; #1-1腔体破真空阈值到达延时（测试）
ANDNOT 801.09  ; #1腔体顶伸气缸下降位标志[0001.09]
OUT D1077.05  ; #1腔体腔体顶升气缸下降（复位）
LD TR0
LD 801.05  ; #1腔体平移一级气缸伸出位标志[0001.05]
AND 801.07  ; #1腔体平移二级气缸伸出位标志[0001.07]
NOT(520)
OR P_On
ANDLD
AND D1062.00  ; #1腔体机构平移气缸安全移动条件
OUT D1077.06  ; #1腔体腔体平移气缸伸出（复位）
; rung 4
ILC(003)

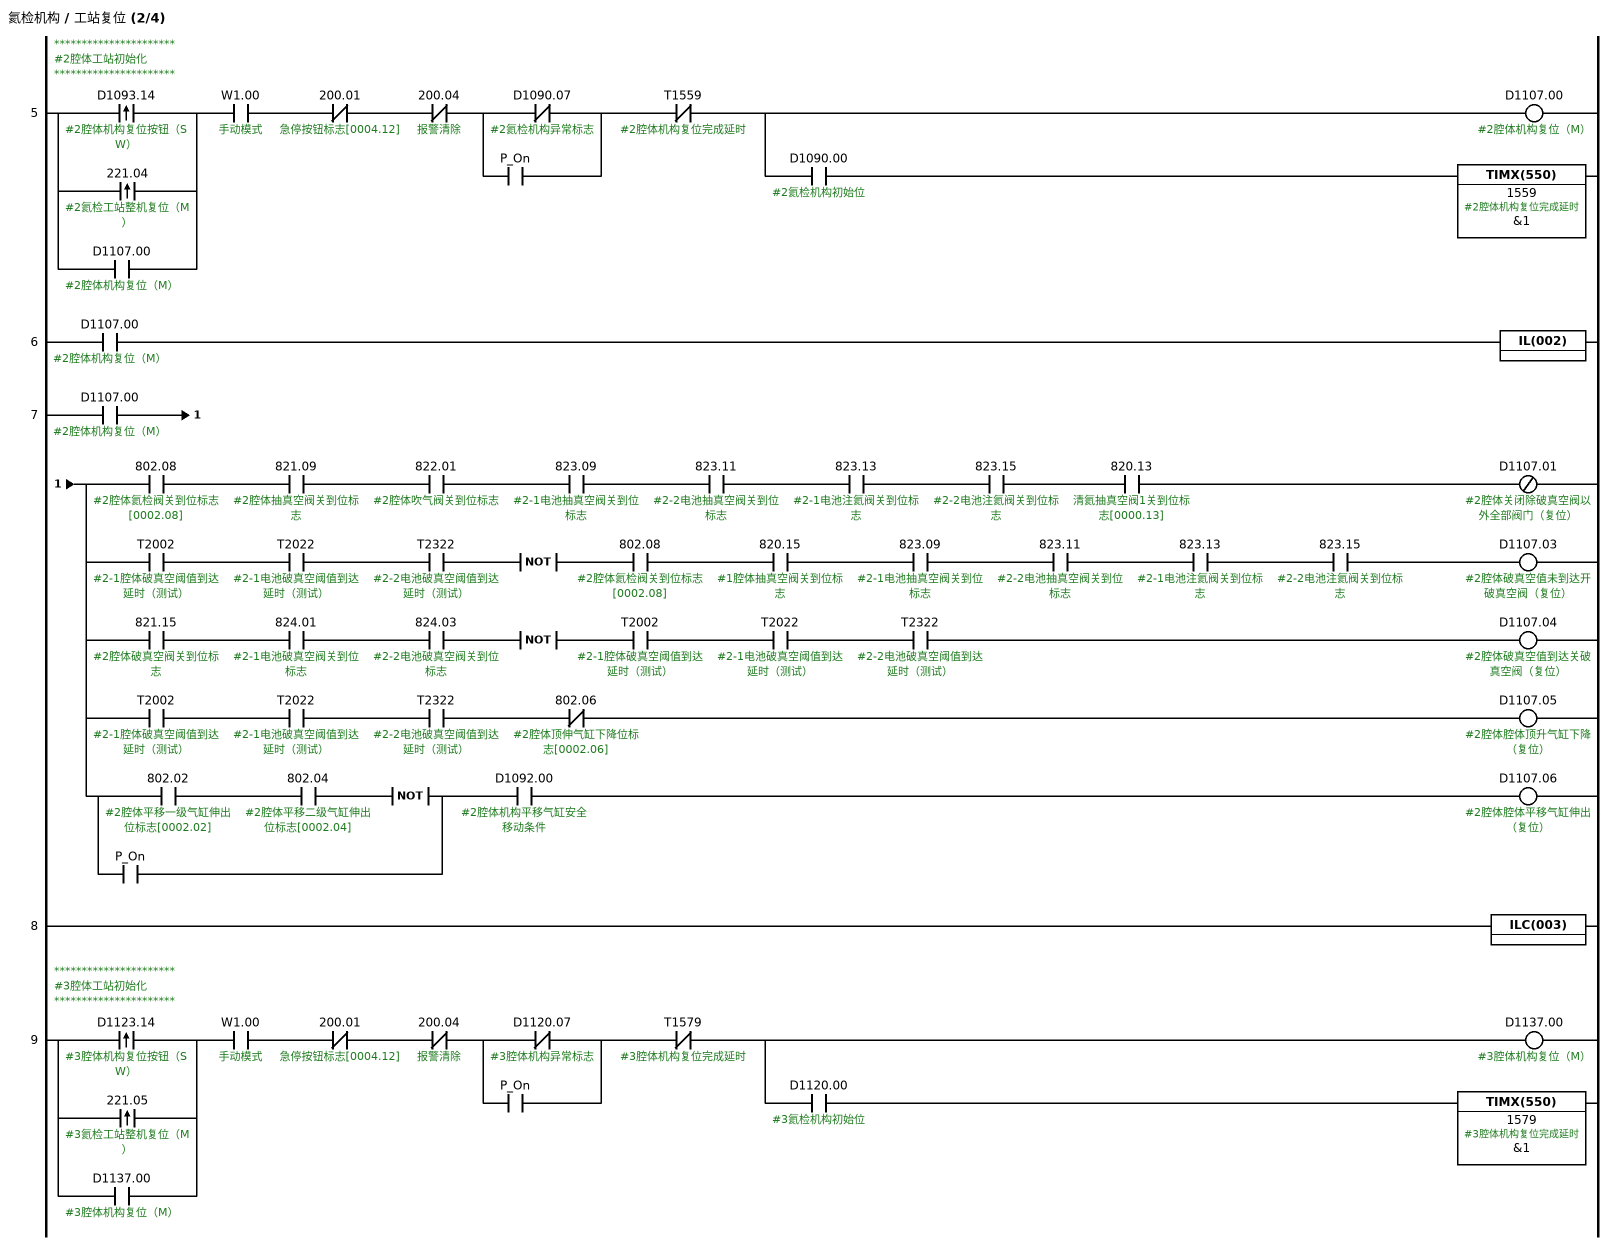
; rung 5: ********************** / #2腔体工站初始化 / **********************
@LD D1093.14  ; #2腔体机构复位按钮（SW）
@OR 221.04  ; #2氦检工站整机复位（M）
OR D1107.00  ; #2腔体机构复位（M）
AND W1.00  ; 手动模式
ANDNOT 200.01  ; 急停按钮标志[0004.12]
ANDNOT 200.04  ; 报警清除
LDNOT D1090.07  ; #2氦检机构异常标志
OR P_On
ANDLD
ANDNOT T1559  ; #2腔体机构复位完成延时
OUT D1107.00  ; #2腔体机构复位（M）
AND D1090.00  ; #2氦检机构初始位
TIMX(550) 1559 &1  ; #2腔体机构复位完成延时
; rung 6
LD D1107.00  ; #2腔体机构复位（M）
IL(002)
; rung 7
LD D1107.00  ; #2腔体机构复位（M）
OUT TR0
AND 802.08  ; #2腔体氦检阀关到位标志[0002.08]
AND 821.09  ; #2腔体抽真空阀关到位标志
AND 822.01  ; #2腔体吹气阀关到位标志
AND 823.09  ; #2-1电池抽真空阀关到位标志
AND 823.11  ; #2-2电池抽真空阀关到位标志
AND 823.13  ; #2-1电池注氦阀关到位标志
AND 823.15  ; #2-2电池注氦阀关到位标志
AND 820.13  ; 清氦抽真空阀1关到位标志[0000.13]
OUTNOT D1107.01  ; #2腔体关闭除破真空阀以外全部阀门（复位）
LD TR0
AND T2002  ; #2-1腔体破真空阈值到达延时（测试）
AND T2022  ; #2-1电池破真空阈值到达延时（测试）
AND T2322  ; #2-2电池破真空阈值到达延时（测试）
NOT(520)
AND 802.08  ; #2腔体氦检阀关到位标志[0002.08]
AND 820.15  ; #1腔体抽真空阀关到位标志
AND 823.09  ; #2-1电池抽真空阀关到位标志
AND 823.11  ; #2-2电池抽真空阀关到位标志
AND 823.13  ; #2-1电池注氦阀关到位标志
AND 823.15  ; #2-2电池注氦阀关到位标志
OUT D1107.03  ; #2腔体破真空值未到达开破真空阀（复位）
LD TR0
AND 821.15  ; #2腔体破真空阀关到位标志
AND 824.01  ; #2-1电池破真空阀关到位标志
AND 824.03  ; #2-2电池破真空阀关到位标志
NOT(520)
AND T2002  ; #2-1腔体破真空阈值到达延时（测试）
AND T2022  ; #2-1电池破真空阈值到达延时（测试）
AND T2322  ; #2-2电池破真空阈值到达延时（测试）
OUT D1107.04  ; #2腔体破真空值到达关破真空阀（复位）
LD TR0
AND T2002  ; #2-1腔体破真空阈值到达延时（测试）
AND T2022  ; #2-1电池破真空阈值到达延时（测试）
AND T2322  ; #2-2电池破真空阈值到达延时（测试）
ANDNOT 802.06  ; #2腔体顶伸气缸下降位标志[0002.06]
OUT D1107.05  ; #2腔体腔体顶升气缸下降（复位）
LD TR0
LD 802.02  ; #2腔体平移一级气缸伸出位标志[0002.02]
AND 802.04  ; #2腔体平移二级气缸伸出位标志[0002.04]
NOT(520)
OR P_On
ANDLD
AND D1092.00  ; #2腔体机构平移气缸安全移动条件
OUT D1107.06  ; #2腔体腔体平移气缸伸出（复位）
; rung 8
ILC(003)
; rung 9: ********************** / #3腔体工站初始化 / **********************
@LD D1123.14  ; #3腔体机构复位按钮（SW）
@OR 221.05  ; #3氦检工站整机复位（M）
OR D1137.00  ; #3腔体机构复位（M）
AND W1.00  ; 手动模式
ANDNOT 200.01  ; 急停按钮标志[0004.12]
ANDNOT 200.04  ; 报警清除
LDNOT D1120.07  ; #3腔体机构异常标志
OR P_On
ANDLD
ANDNOT T1579  ; #3腔体机构复位完成延时
OUT D1137.00  ; #3腔体机构复位（M）
AND D1120.00  ; #3氦检机构初始位
TIMX(550) 1579 &1  ; #3腔体机构复位完成延时

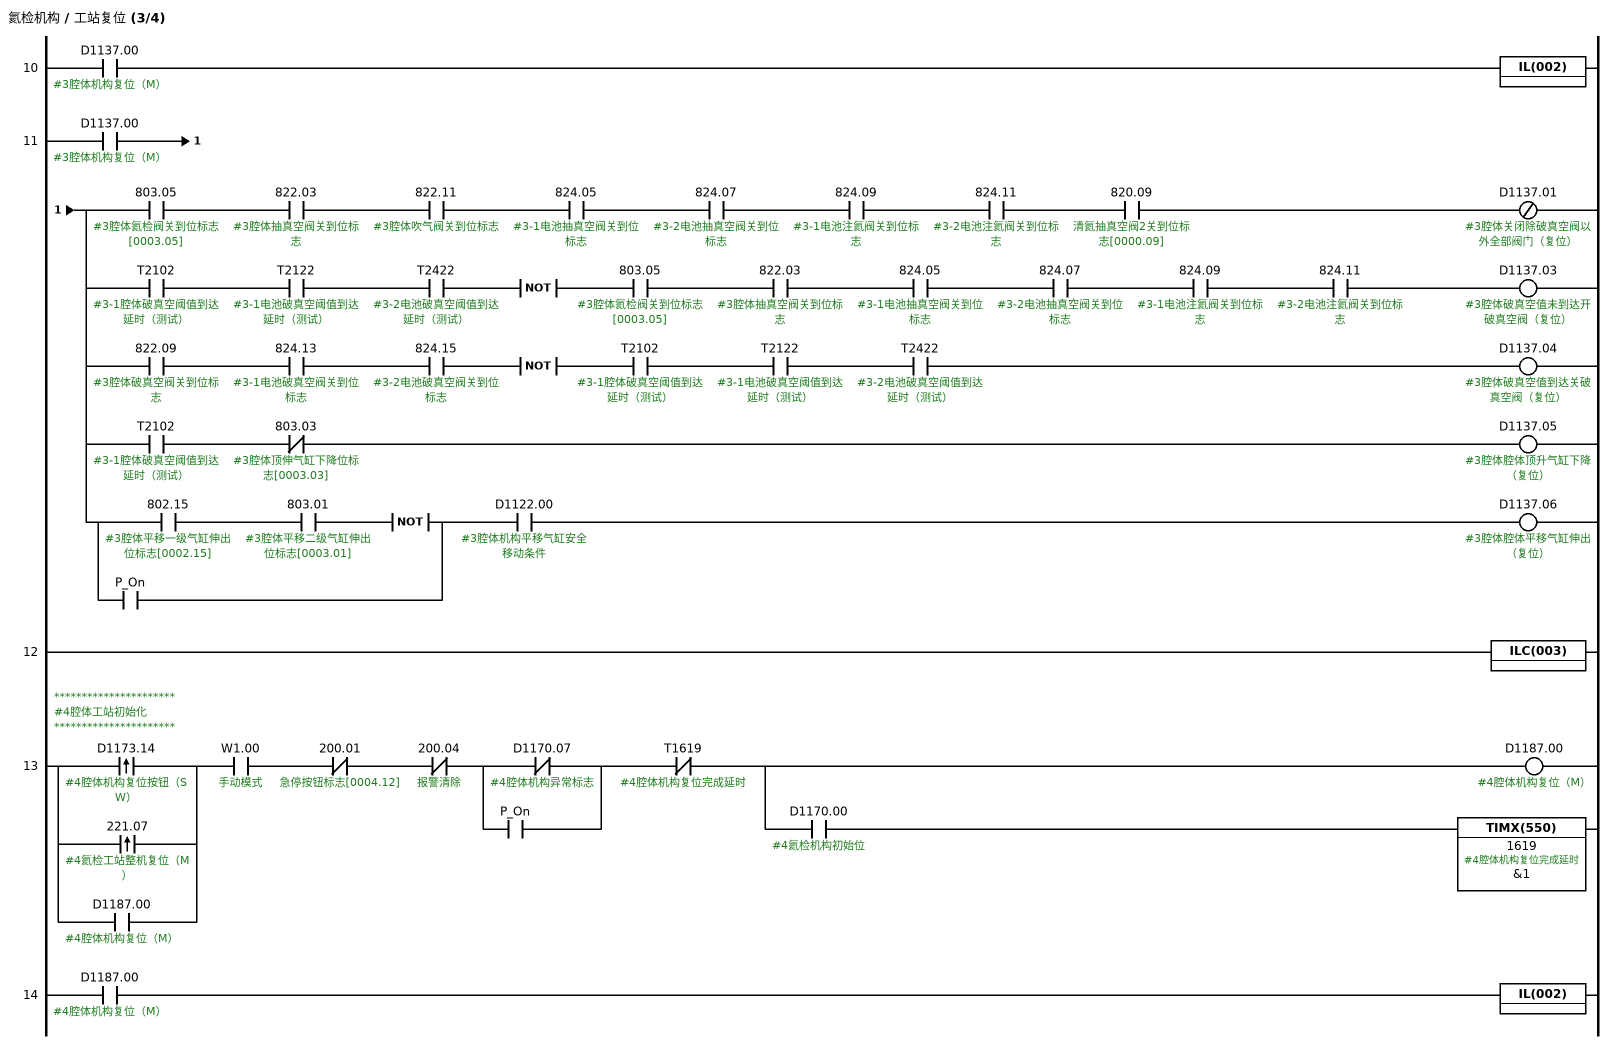
; rung 10
LD D1137.00  ; #3腔体机构复位（M）
IL(002)
; rung 11
LD D1137.00  ; #3腔体机构复位（M）
OUT TR0
AND 803.05  ; #3腔体氦检阀关到位标志[0003.05]
AND 822.03  ; #3腔体抽真空阀关到位标志
AND 822.11  ; #3腔体吹气阀关到位标志
AND 824.05  ; #3-1电池抽真空阀关到位标志
AND 824.07  ; #3-2电池抽真空阀关到位标志
AND 824.09  ; #3-1电池注氦阀关到位标志
AND 824.11  ; #3-2电池注氦阀关到位标志
AND 820.09  ; 清氦抽真空阀2关到位标志[0000.09]
OUTNOT D1137.01  ; #3腔体关闭除破真空阀以外全部阀门（复位）
LD TR0
AND T2102  ; #3-1腔体破真空阈值到达延时（测试）
AND T2122  ; #3-1电池破真空阈值到达延时（测试）
AND T2422  ; #3-2电池破真空阈值到达延时（测试）
NOT(520)
AND 803.05  ; #3腔体氦检阀关到位标志[0003.05]
AND 822.03  ; #3腔体抽真空阀关到位标志
AND 824.05  ; #3-1电池抽真空阀关到位标志
AND 824.07  ; #3-2电池抽真空阀关到位标志
AND 824.09  ; #3-1电池注氦阀关到位标志
AND 824.11  ; #3-2电池注氦阀关到位标志
OUT D1137.03  ; #3腔体破真空值未到达开破真空阀（复位）
LD TR0
AND 822.09  ; #3腔体破真空阀关到位标志
AND 824.13  ; #3-1电池破真空阀关到位标志
AND 824.15  ; #3-2电池破真空阀关到位标志
NOT(520)
AND T2102  ; #3-1腔体破真空阈值到达延时（测试）
AND T2122  ; #3-1电池破真空阈值到达延时（测试）
AND T2422  ; #3-2电池破真空阈值到达延时（测试）
OUT D1137.04  ; #3腔体破真空值到达关破真空阀（复位）
LD TR0
AND T2102  ; #3-1腔体破真空阈值到达延时（测试）
ANDNOT 803.03  ; #3腔体顶伸气缸下降位标志[0003.03]
OUT D1137.05  ; #3腔体腔体顶升气缸下降（复位）
LD TR0
LD 802.15  ; #3腔体平移一级气缸伸出位标志[0002.15]
AND 803.01  ; #3腔体平移二级气缸伸出位标志[0003.01]
NOT(520)
OR P_On
ANDLD
AND D1122.00  ; #3腔体机构平移气缸安全移动条件
OUT D1137.06  ; #3腔体腔体平移气缸伸出（复位）
; rung 12
ILC(003)
; rung 13: ********************** / #4腔体工站初始化 / **********************
@LD D1173.14  ; #4腔体机构复位按钮（SW）
@OR 221.07  ; #4氦检工站整机复位（M）
OR D1187.00  ; #4腔体机构复位（M）
AND W1.00  ; 手动模式
ANDNOT 200.01  ; 急停按钮标志[0004.12]
ANDNOT 200.04  ; 报警清除
LDNOT D1170.07  ; #4腔体机构异常标志
OR P_On
ANDLD
ANDNOT T1619  ; #4腔体机构复位完成延时
OUT D1187.00  ; #4腔体机构复位（M）
AND D1170.00  ; #4氦检机构初始位
TIMX(550) 1619 &1  ; #4腔体机构复位完成延时
; rung 14
LD D1187.00  ; #4腔体机构复位（M）
IL(002)

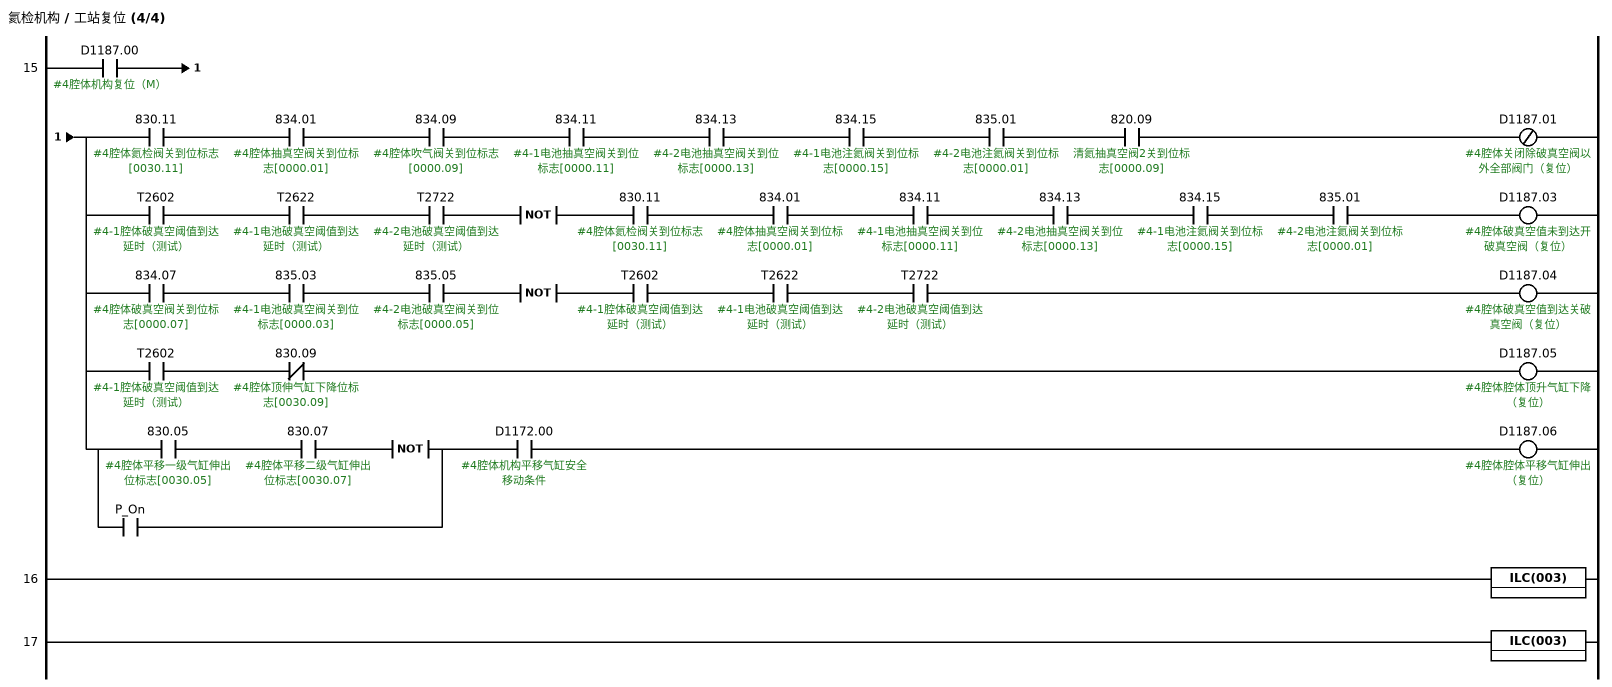
; rung 15
LD D1187.00  ; #4腔体机构复位（M）
OUT TR0
AND 830.11  ; #4腔体氦检阀关到位标志[0030.11]
AND 834.01  ; #4腔体抽真空阀关到位标志[0000.01]
AND 834.09  ; #4腔体吹气阀关到位标志[0000.09]
AND 834.11  ; #4-1电池抽真空阀关到位标志[0000.11]
AND 834.13  ; #4-2电池抽真空阀关到位标志[0000.13]
AND 834.15  ; #4-1电池注氦阀关到位标志[0000.15]
AND 835.01  ; #4-2电池注氦阀关到位标志[0000.01]
AND 820.09  ; 清氦抽真空阀2关到位标志[0000.09]
OUTNOT D1187.01  ; #4腔体关闭除破真空阀以外全部阀门（复位）
LD TR0
AND T2602  ; #4-1腔体破真空阈值到达延时（测试）
AND T2622  ; #4-1电池破真空阈值到达延时（测试）
AND T2722  ; #4-2电池破真空阈值到达延时（测试）
NOT(520)
AND 830.11  ; #4腔体氦检阀关到位标志[0030.11]
AND 834.01  ; #4腔体抽真空阀关到位标志[0000.01]
AND 834.11  ; #4-1电池抽真空阀关到位标志[0000.11]
AND 834.13  ; #4-2电池抽真空阀关到位标志[0000.13]
AND 834.15  ; #4-1电池注氦阀关到位标志[0000.15]
AND 835.01  ; #4-2电池注氦阀关到位标志[0000.01]
OUT D1187.03  ; #4腔体破真空值未到达开破真空阀（复位）
LD TR0
AND 834.07  ; #4腔体破真空阀关到位标志[0000.07]
AND 835.03  ; #4-1电池破真空阀关到位标志[0000.03]
AND 835.05  ; #4-2电池破真空阀关到位标志[0000.05]
NOT(520)
AND T2602  ; #4-1腔体破真空阈值到达延时（测试）
AND T2622  ; #4-1电池破真空阈值到达延时（测试）
AND T2722  ; #4-2电池破真空阈值到达延时（测试）
OUT D1187.04  ; #4腔体破真空值到达关破真空阀（复位）
LD TR0
AND T2602  ; #4-1腔体破真空阈值到达延时（测试）
ANDNOT 830.09  ; #4腔体顶伸气缸下降位标志[0030.09]
OUT D1187.05  ; #4腔体腔体顶升气缸下降（复位）
LD TR0
LD 830.05  ; #4腔体平移一级气缸伸出位标志[0030.05]
AND 830.07  ; #4腔体平移二级气缸伸出位标志[0030.07]
NOT(520)
OR P_On
ANDLD
AND D1172.00  ; #4腔体机构平移气缸安全移动条件
OUT D1187.06  ; #4腔体腔体平移气缸伸出（复位）
; rung 16
ILC(003)
; rung 17
ILC(003)

### Section 腔体标漏

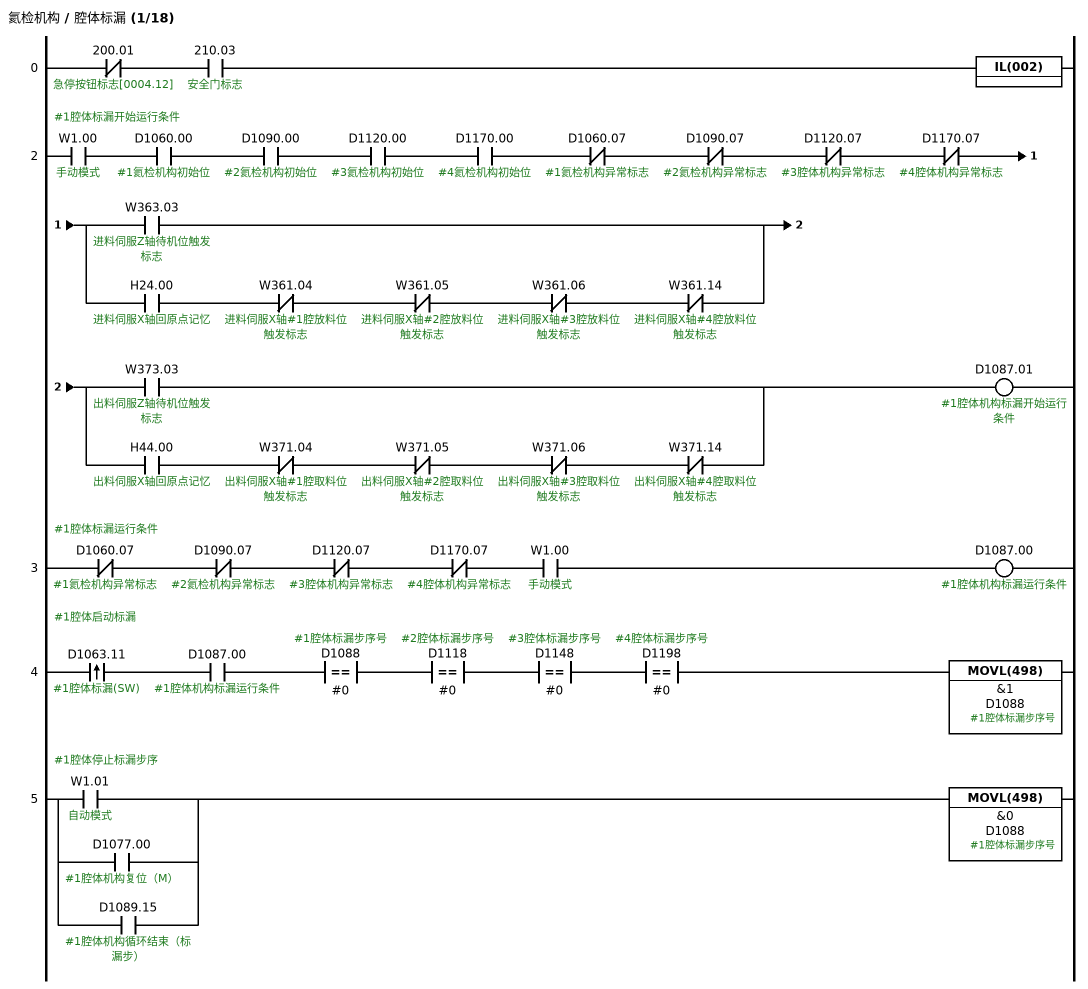
; rung 0
LDNOT 200.01  ; 急停按钮标志[0004.12]
AND 210.03  ; 安全门标志
IL(002)
; rung 1: ********************** / #1腔体标漏流程 / **********************
; rung 2: #1腔体标漏开始运行条件
LD W1.00  ; 手动模式
AND D1060.00  ; #1氦检机构初始位
AND D1090.00  ; #2氦检机构初始位
AND D1120.00  ; #3氦检机构初始位
AND D1170.00  ; #4氦检机构初始位
ANDNOT D1060.07  ; #1氦检机构异常标志
ANDNOT D1090.07  ; #2氦检机构异常标志
ANDNOT D1120.07  ; #3腔体机构异常标志
ANDNOT D1170.07  ; #4腔体机构异常标志
LD W363.03  ; 进料伺服Z轴待机位触发标志
LD H24.00  ; 进料伺服X轴回原点记忆
ANDNOT W361.04  ; 进料伺服X轴#1腔放料位触发标志
ANDNOT W361.05  ; 进料伺服X轴#2腔放料位触发标志
ANDNOT W361.06  ; 进料伺服X轴#3腔放料位触发标志
ANDNOT W361.14  ; 进料伺服X轴#4腔放料位触发标志
ORLD
ANDLD
LD W373.03  ; 出料伺服Z轴待机位触发标志
LD H44.00  ; 出料伺服X轴回原点记忆
ANDNOT W371.04  ; 出料伺服X轴#1腔取料位触发标志
ANDNOT W371.05  ; 出料伺服X轴#2腔取料位触发标志
ANDNOT W371.06  ; 出料伺服X轴#3腔取料位触发标志
ANDNOT W371.14  ; 出料伺服X轴#4腔取料位触发标志
ORLD
ANDLD
OUT D1087.01  ; #1腔体机构标漏开始运行条件
; rung 3: #1腔体标漏运行条件
LDNOT D1060.07  ; #1氦检机构异常标志
ANDNOT D1090.07  ; #2氦检机构异常标志
ANDNOT D1120.07  ; #3腔体机构异常标志
ANDNOT D1170.07  ; #4腔体机构异常标志
AND W1.00  ; 手动模式
OUT D1087.00  ; #1腔体机构标漏运行条件
; rung 4: #1腔体启动标漏
@LD D1063.11  ; #1腔体标漏(SW)
AND D1087.00  ; #1腔体机构标漏运行条件
AND=L(301) D1088 #0  ; #1腔体标漏步序号
AND=L(301) D1118 #0  ; #2腔体标漏步序号
AND=L(301) D1148 #0  ; #3腔体标漏步序号
AND=L(301) D1198 #0  ; #4腔体标漏步序号
MOVL(498) &1 D1088  ; #1腔体标漏步序号
; rung 5: #1腔体停止标漏步序
LD W1.01  ; 自动模式
OR D1077.00  ; #1腔体机构复位（M）
OR D1089.15  ; #1腔体机构循环结束（标漏步）
MOVL(498) &0 D1088  ; #1腔体标漏步序号

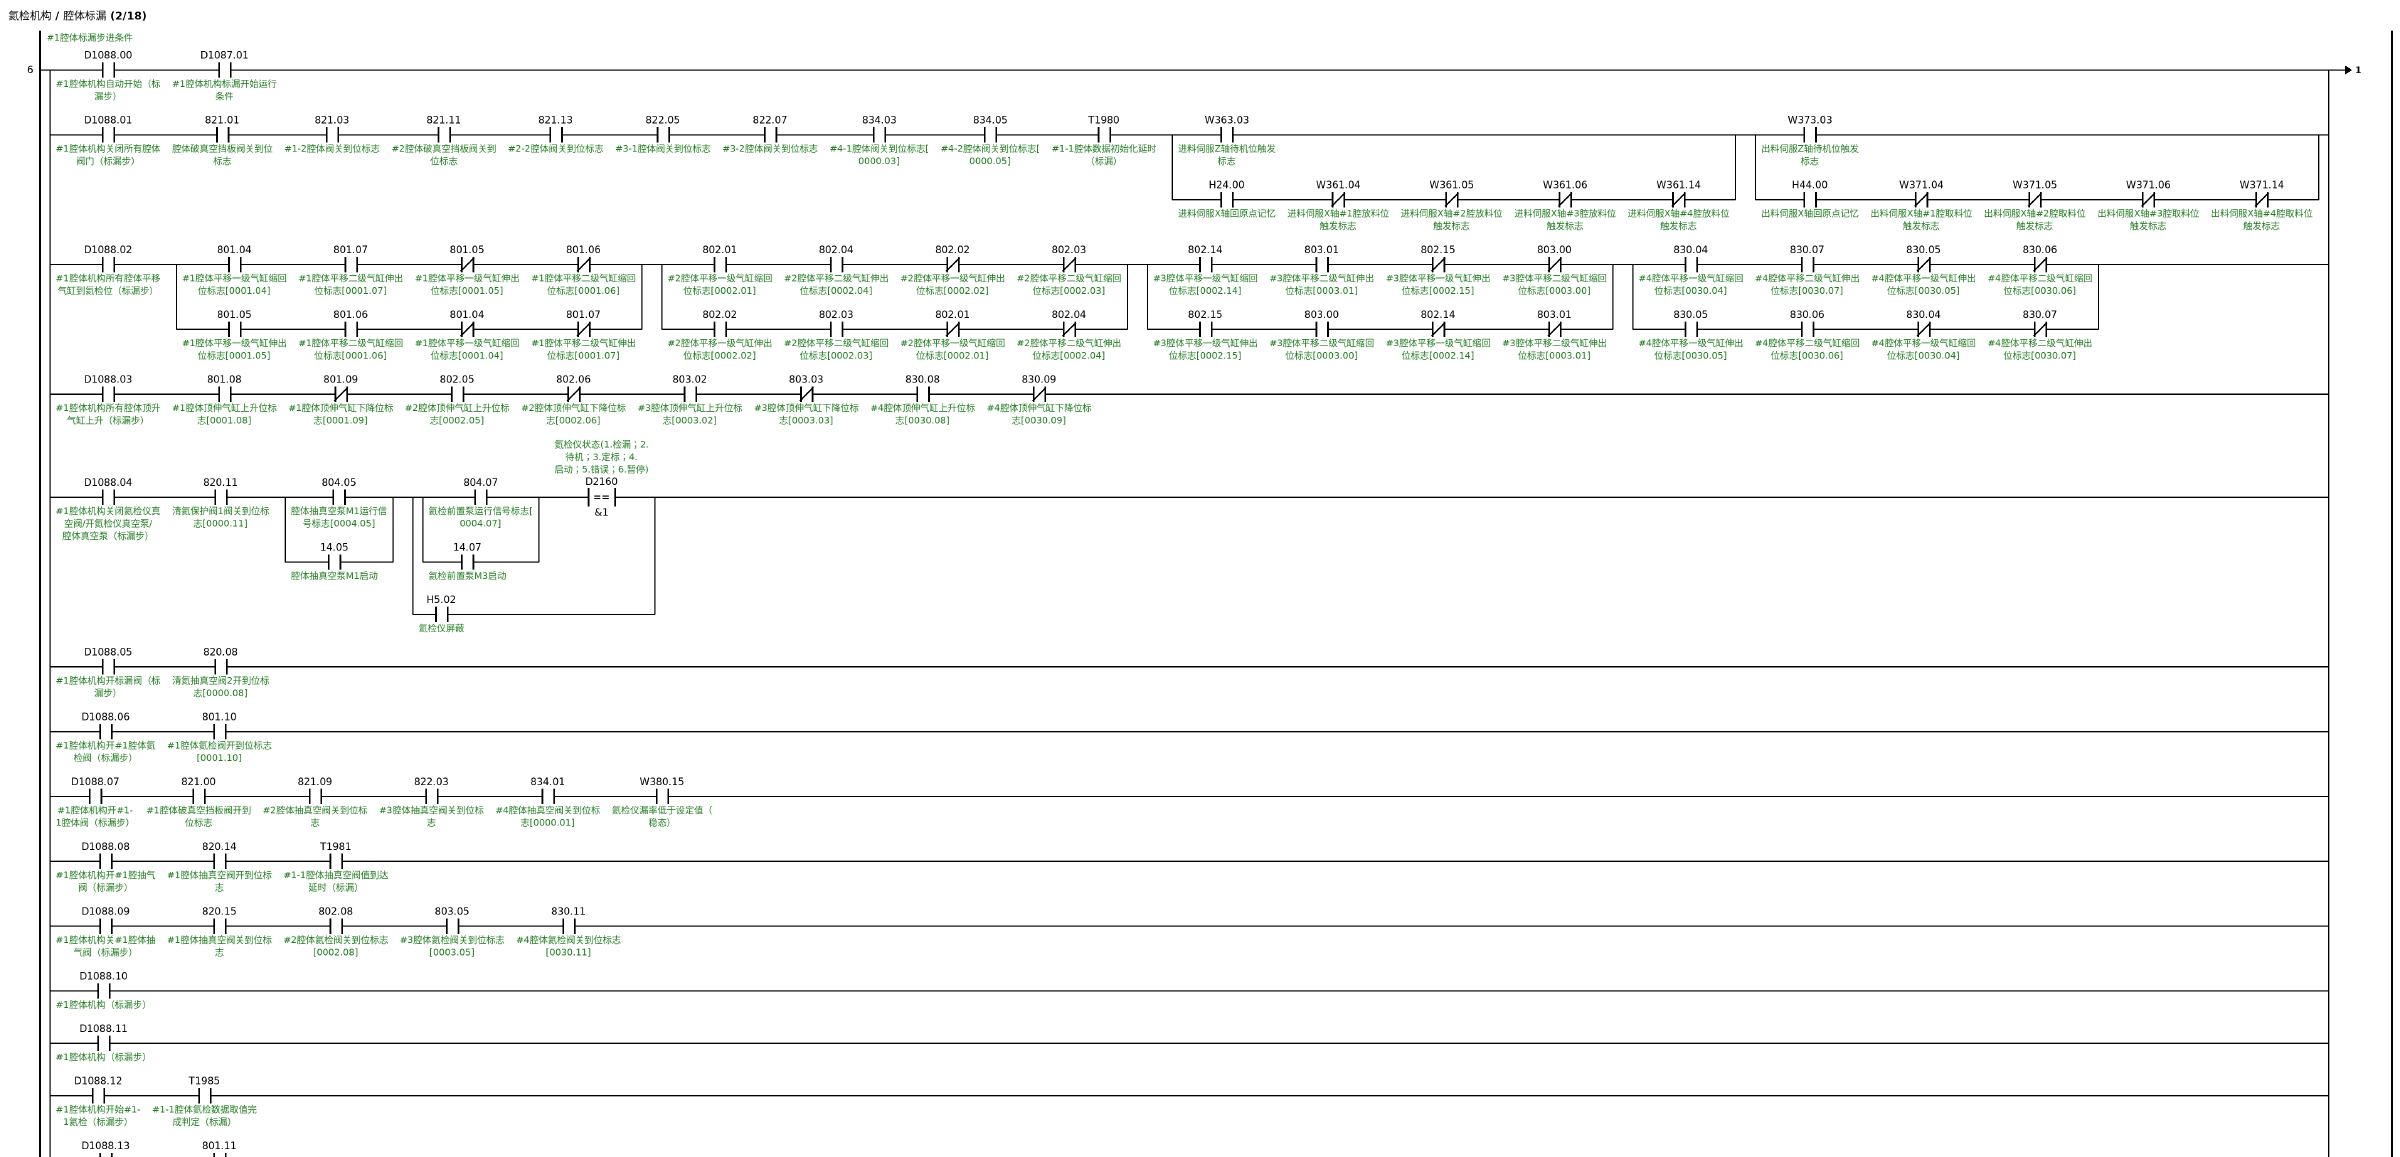

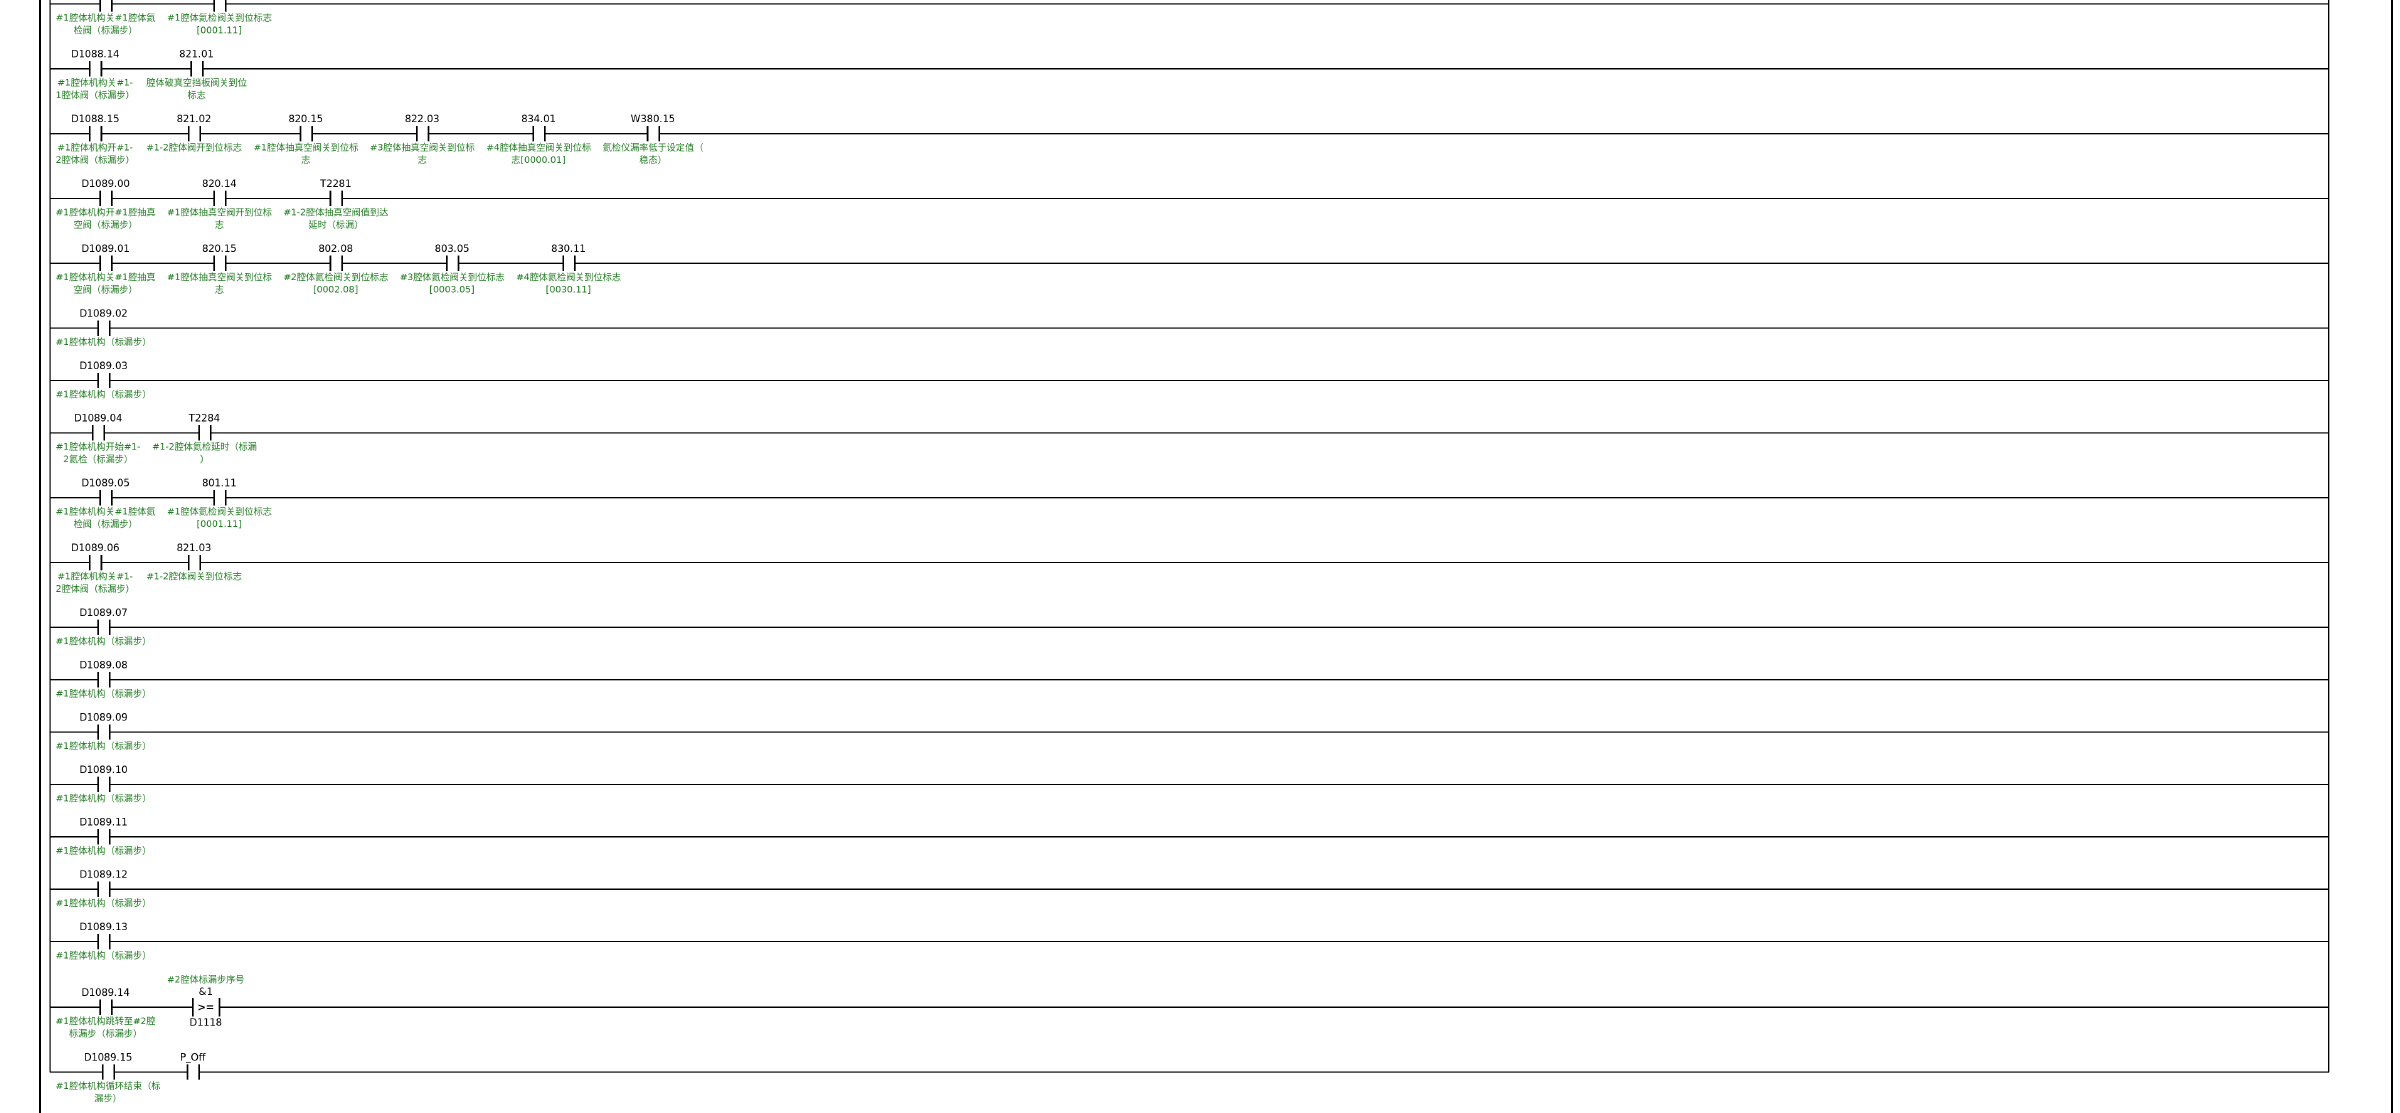

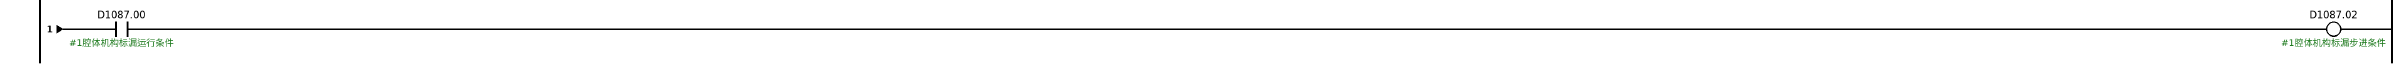
; rung 6: #1腔体标漏步进条件
LD D1088.00  ; #1腔体机构自动开始（标漏步）
AND D1087.01  ; #1腔体机构标漏开始运行条件
LD D1088.01  ; #1腔体机构关闭所有腔体阀门（标漏步）
AND 821.01  ; 腔体破真空挡板阀关到位标志
AND 821.03  ; #1-2腔体阀关到位标志
AND 821.11  ; #2腔体破真空挡板阀关到位标志
AND 821.13  ; #2-2腔体阀关到位标志
AND 822.05  ; #3-1腔体阀关到位标志
AND 822.07  ; #3-2腔体阀关到位标志
AND 834.03  ; #4-1腔体阀关到位标志[0000.03]
AND 834.05  ; #4-2腔体阀关到位标志[0000.05]
AND T1980  ; #1-1腔体数据初始化延时（标漏）
LD W363.03  ; 进料伺服Z轴待机位触发标志
LD H24.00  ; 进料伺服X轴回原点记忆
ANDNOT W361.04  ; 进料伺服X轴#1腔放料位触发标志
ANDNOT W361.05  ; 进料伺服X轴#2腔放料位触发标志
ANDNOT W361.06  ; 进料伺服X轴#3腔放料位触发标志
ANDNOT W361.14  ; 进料伺服X轴#4腔放料位触发标志
ORLD
ANDLD
LD W373.03  ; 出料伺服Z轴待机位触发标志
LD H44.00  ; 出料伺服X轴回原点记忆
ANDNOT W371.04  ; 出料伺服X轴#1腔取料位触发标志
ANDNOT W371.05  ; 出料伺服X轴#2腔取料位触发标志
ANDNOT W371.06  ; 出料伺服X轴#3腔取料位触发标志
ANDNOT W371.14  ; 出料伺服X轴#4腔取料位触发标志
ORLD
ANDLD
ORLD
LD D1088.02  ; #1腔体机构所有腔体平移气缸到氦检位（标漏步）
LD 801.04  ; #1腔体平移一级气缸缩回位标志[0001.04]
AND 801.07  ; #1腔体平移二级气缸伸出位标志[0001.07]
ANDNOT 801.05  ; #1腔体平移一级气缸伸出位标志[0001.05]
ANDNOT 801.06  ; #1腔体平移二级气缸缩回位标志[0001.06]
LD 801.05  ; #1腔体平移一级气缸伸出位标志[0001.05]
AND 801.06  ; #1腔体平移二级气缸缩回位标志[0001.06]
ANDNOT 801.04  ; #1腔体平移一级气缸缩回位标志[0001.04]
ANDNOT 801.07  ; #1腔体平移二级气缸伸出位标志[0001.07]
ORLD
ANDLD
LD 802.01  ; #2腔体平移一级气缸缩回位标志[0002.01]
AND 802.04  ; #2腔体平移二级气缸伸出位标志[0002.04]
ANDNOT 802.02  ; #2腔体平移一级气缸伸出位标志[0002.02]
ANDNOT 802.03  ; #2腔体平移二级气缸缩回位标志[0002.03]
LD 802.02  ; #2腔体平移一级气缸伸出位标志[0002.02]
AND 802.03  ; #2腔体平移二级气缸缩回位标志[0002.03]
ANDNOT 802.01  ; #2腔体平移一级气缸缩回位标志[0002.01]
ANDNOT 802.04  ; #2腔体平移二级气缸伸出位标志[0002.04]
ORLD
ANDLD
LD 802.14  ; #3腔体平移一级气缸缩回位标志[0002.14]
AND 803.01  ; #3腔体平移二级气缸伸出位标志[0003.01]
ANDNOT 802.15  ; #3腔体平移一级气缸伸出位标志[0002.15]
ANDNOT 803.00  ; #3腔体平移二级气缸缩回位标志[0003.00]
LD 802.15  ; #3腔体平移一级气缸伸出位标志[0002.15]
AND 803.00  ; #3腔体平移二级气缸缩回位标志[0003.00]
ANDNOT 802.14  ; #3腔体平移一级气缸缩回位标志[0002.14]
ANDNOT 803.01  ; #3腔体平移二级气缸伸出位标志[0003.01]
ORLD
ANDLD
LD 830.04  ; #4腔体平移一级气缸缩回位标志[0030.04]
AND 830.07  ; #4腔体平移二级气缸伸出位标志[0030.07]
ANDNOT 830.05  ; #4腔体平移一级气缸伸出位标志[0030.05]
ANDNOT 830.06  ; #4腔体平移二级气缸缩回位标志[0030.06]
LD 830.05  ; #4腔体平移一级气缸伸出位标志[0030.05]
AND 830.06  ; #4腔体平移二级气缸缩回位标志[0030.06]
ANDNOT 830.04  ; #4腔体平移一级气缸缩回位标志[0030.04]
ANDNOT 830.07  ; #4腔体平移二级气缸伸出位标志[0030.07]
ORLD
ANDLD
ORLD
LD D1088.03  ; #1腔体机构所有腔体顶升气缸上升（标漏步）
AND 801.08  ; #1腔体顶伸气缸上升位标志[0001.08]
ANDNOT 801.09  ; #1腔体顶伸气缸下降位标志[0001.09]
AND 802.05  ; #2腔体顶伸气缸上升位标志[0002.05]
ANDNOT 802.06  ; #2腔体顶伸气缸下降位标志[0002.06]
AND 803.02  ; #3腔体顶伸气缸上升位标志[0003.02]
ANDNOT 803.03  ; #3腔体顶伸气缸下降位标志[0003.03]
AND 830.08  ; #4腔体顶伸气缸上升位标志[0030.08]
ANDNOT 830.09  ; #4腔体顶伸气缸下降位标志[0030.09]
ORLD
LD D1088.04  ; #1腔体机构关闭氦检仪真空阀/开氦检仪真空泵/腔体真空泵（标漏步）
AND 820.11  ; 清氦保护阀1阀关到位标志[0000.11]
LD 804.05  ; 腔体抽真空泵M1运行信号标志[0004.05]
OR 14.05  ; 腔体抽真空泵M1启动
ANDLD
LD 804.07  ; 氦检前置泵运行信号标志[0004.07]
OR 14.07  ; 氦检前置泵M3启动
AND=(300) D2160 &1  ; 氦检仪状态(1.检漏；2.待机；3.定标；4.启动；5.错误；6.暂停)
OR H5.02  ; 氦检仪屏蔽
ANDLD
ORLD
LD D1088.05  ; #1腔体机构开标漏阀（标漏步）
AND 820.08  ; 清氦抽真空阀2开到位标志[0000.08]
ORLD
LD D1088.06  ; #1腔体机构开#1腔体氦检阀（标漏步）
AND 801.10  ; #1腔体氦检阀开到位标志[0001.10]
ORLD
LD D1088.07  ; #1腔体机构开#1-1腔体阀（标漏步）
AND 821.00  ; #1腔体破真空挡板阀开到位标志
AND 821.09  ; #2腔体抽真空阀关到位标志
AND 822.03  ; #3腔体抽真空阀关到位标志
AND 834.01  ; #4腔体抽真空阀关到位标志[0000.01]
AND W380.15  ; 氦检仪漏率低于设定值（稳态）
ORLD
LD D1088.08  ; #1腔体机构开#1腔抽气阀（标漏步）
AND 820.14  ; #1腔体抽真空阀开到位标志
AND T1981  ; #1-1腔体抽真空阀值到达延时（标漏）
ORLD
LD D1088.09  ; #1腔体机构关#1腔体抽气阀（标漏步）
AND 820.15  ; #1腔体抽真空阀关到位标志
AND 802.08  ; #2腔体氦检阀关到位标志[0002.08]
AND 803.05  ; #3腔体氦检阀关到位标志[0003.05]
AND 830.11  ; #4腔体氦检阀关到位标志[0030.11]
ORLD
OR D1088.10  ; #1腔体机构（标漏步）
OR D1088.11  ; #1腔体机构（标漏步）
LD D1088.12  ; #1腔体机构开始#1-1氦检（标漏步）
AND T1985  ; #1-1腔体氦检数据取值完成判定（标漏）
ORLD
LD D1088.13  ; #1腔体机构关#1腔体氦检阀（标漏步）
AND 801.11  ; #1腔体氦检阀关到位标志[0001.11]
ORLD
LD D1088.14  ; #1腔体机构关#1-1腔体阀（标漏步）
AND 821.01  ; 腔体破真空挡板阀关到位标志
ORLD
LD D1088.15  ; #1腔体机构开#1-2腔体阀（标漏步）
AND 821.02  ; #1-2腔体阀开到位标志
AND 820.15  ; #1腔体抽真空阀关到位标志
AND 822.03  ; #3腔体抽真空阀关到位标志
AND 834.01  ; #4腔体抽真空阀关到位标志[0000.01]
AND W380.15  ; 氦检仪漏率低于设定值（稳态）
ORLD
LD D1089.00  ; #1腔体机构开#1腔抽真空阀（标漏步）
AND 820.14  ; #1腔体抽真空阀开到位标志
AND T2281  ; #1-2腔体抽真空阀值到达延时（标漏）
ORLD
LD D1089.01  ; #1腔体机构关#1腔抽真空阀（标漏步）
AND 820.15  ; #1腔体抽真空阀关到位标志
AND 802.08  ; #2腔体氦检阀关到位标志[0002.08]
AND 803.05  ; #3腔体氦检阀关到位标志[0003.05]
AND 830.11  ; #4腔体氦检阀关到位标志[0030.11]
ORLD
OR D1089.02  ; #1腔体机构（标漏步）
OR D1089.03  ; #1腔体机构（标漏步）
LD D1089.04  ; #1腔体机构开始#1-2氦检（标漏步）
AND T2284  ; #1-2腔体氦检延时（标漏）
ORLD
LD D1089.05  ; #1腔体机构关#1腔体氦检阀（标漏步）
AND 801.11  ; #1腔体氦检阀关到位标志[0001.11]
ORLD
LD D1089.06  ; #1腔体机构关#1-2腔体阀（标漏步）
AND 821.03  ; #1-2腔体阀关到位标志
ORLD
OR D1089.07  ; #1腔体机构（标漏步）
OR D1089.08  ; #1腔体机构（标漏步）
OR D1089.09  ; #1腔体机构（标漏步）
OR D1089.10  ; #1腔体机构（标漏步）
OR D1089.11  ; #1腔体机构（标漏步）
OR D1089.12  ; #1腔体机构（标漏步）
OR D1089.13  ; #1腔体机构（标漏步）
LD D1089.14  ; #1腔体机构跳转至#2腔标漏步（标漏步）
AND>=L(326) &1 D1118  ; #2腔体标漏步序号
ORLD
LD D1089.15  ; #1腔体机构循环结束（标漏步）
AND P_Off
ORLD
AND D1087.00  ; #1腔体机构标漏运行条件
OUT D1087.02  ; #1腔体机构标漏步进条件

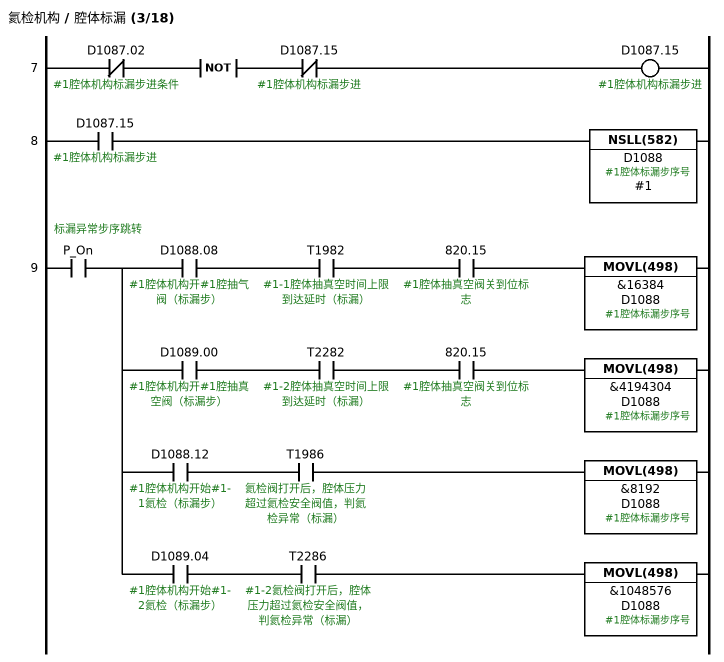
; rung 7
LDNOT D1087.02  ; #1腔体机构标漏步进条件
NOT(520)
ANDNOT D1087.15  ; #1腔体机构标漏步进
OUT D1087.15  ; #1腔体机构标漏步进
; rung 8
LD D1087.15  ; #1腔体机构标漏步进
NSLL(582) D1088 #1  ; #1腔体标漏步序号
; rung 9: 标漏异常步序跳转
LD P_On
OUT TR0
AND D1088.08  ; #1腔体机构开#1腔抽气阀（标漏步）
AND T1982  ; #1-1腔体抽真空时间上限到达延时（标漏）
AND 820.15  ; #1腔体抽真空阀关到位标志
MOVL(498) &16384 D1088  ; #1腔体标漏步序号
LD TR0
AND D1089.00  ; #1腔体机构开#1腔抽真空阀（标漏步）
AND T2282  ; #1-2腔体抽真空时间上限到达延时（标漏）
AND 820.15  ; #1腔体抽真空阀关到位标志
MOVL(498) &4194304 D1088  ; #1腔体标漏步序号
LD TR0
AND D1088.12  ; #1腔体机构开始#1-1氦检（标漏步）
AND T1986  ; 氦检阀打开后，腔体压力超过氦检安全阀值，判氦检异常（标漏）
MOVL(498) &8192 D1088  ; #1腔体标漏步序号
LD TR0
AND D1089.04  ; #1腔体机构开始#1-2氦检（标漏步）
AND T2286  ; #1-2氦检阀打开后，腔体压力超过氦检安全阀值，判氦检异常（标漏）
MOVL(498) &1048576 D1088  ; #1腔体标漏步序号

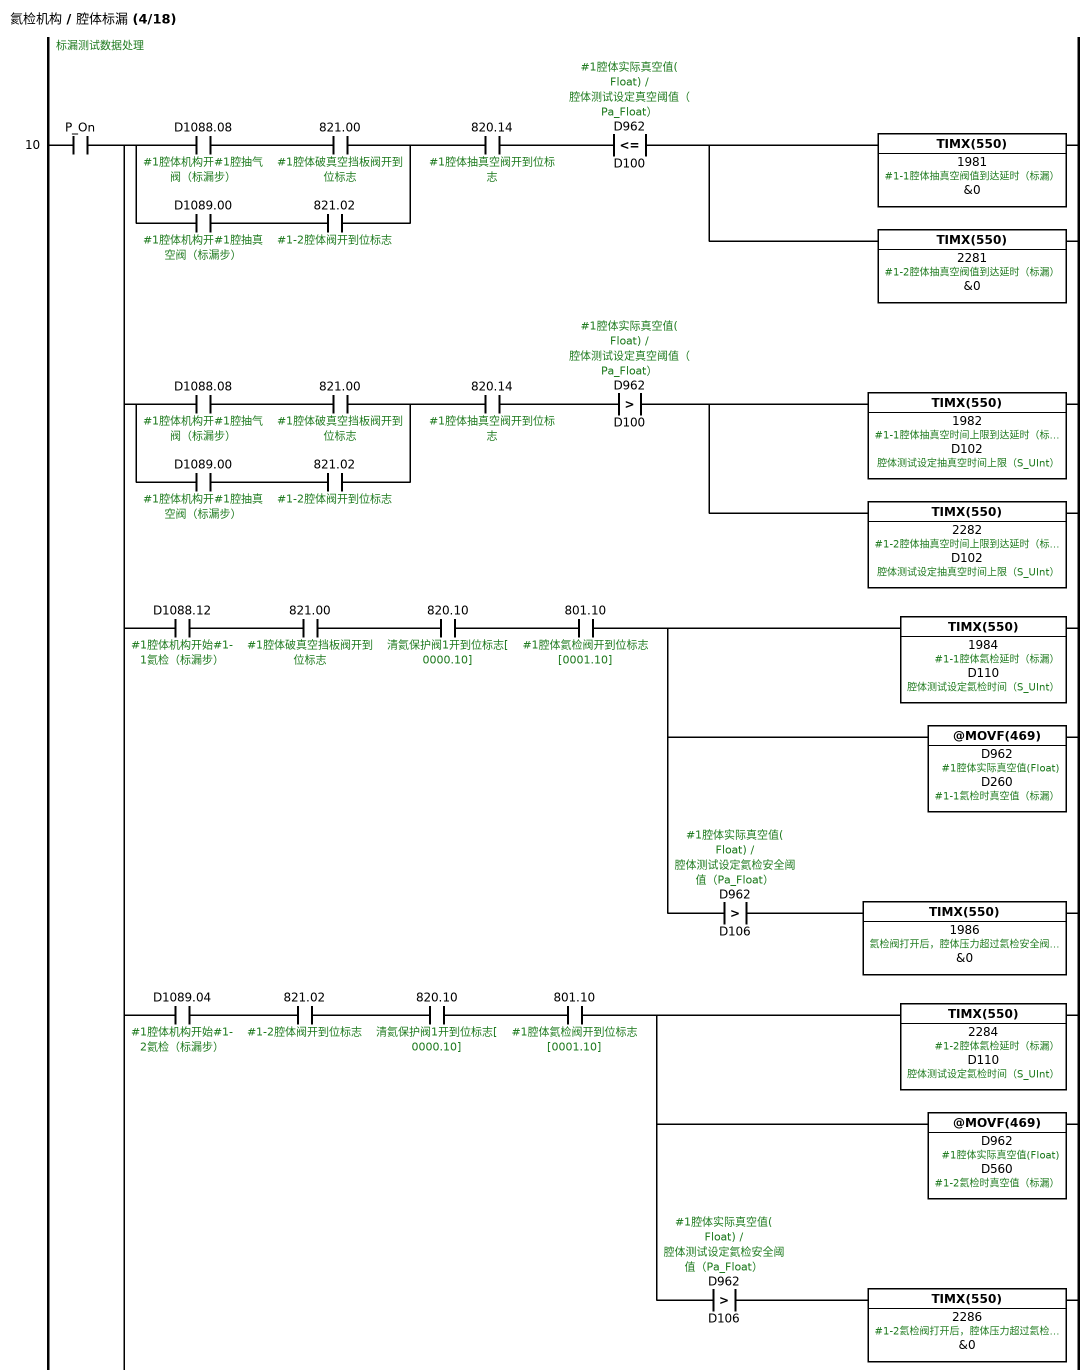

